//CasePacker.Status.Rate.Target := LREAL_TO_INT(csp_main_motorization_manager.motm.actual_velocity_setpoint);
//CasePacker.Status.Rate.Actual := LREAL_TO_INT(csp_main_motorization_manager.motm.actual_velocity);

//CasePacker.Status.Stop.AutoReason := csp_main_interface.alarm_id; 
//CasePacker.Status.Stop.Estop := machine_is_stop_emergency_active(csp.mch);
//CasePacker.Status.Stop.Guard := NOT safety_integrated_series_is_safely_closed(csp_case_main_safety_guards.sis) OR NOT safety_integrated_series_is_safely_closed(csp_transfer_main_safety_guards.sis);
//CasePacker.Status.Stop.Operator := message_is_on(csp_case_main_services_pushbuttons.stop_dchk.alarm_asm.message);

//CasePacker.Status.Starved.CaseBlanks := message_is_on(csp_case_feed_magazine_level_zonemin.magazine_level_zone_min_wem);
//CasePacker.Status.Starved.Glue := NOT digital_input_is_active(csp_case_glue_hotmelt.level_ok_di);
//CasePacker.Status.Starved.Labels :=
//CasePacker.Status.Starved.Units := csp_transfer_infeed_clamp.min_prime;

//CasePacker.Status.Blocked.Downstream := message_is_on(csp_case_discharge_reject_sensors.downstream_backup_hold_aem);
//CasePacker.Status.Blocked.Reject := message_is_on(csp_case_discharge_reject_sensors.consecutive_blocked_reject_aem);
//CasePacker.Status.Blocked.Waste := message_is_on(csp_transfer_crosspusher_reject.backup_di_dchk.alarm_asm.message);

//CasePacker.Labels.Consumed:=


(************************************************************************)

_handle_messages();

_write_output();

ACTION _handle_messages:
;
END_ACTION

ACTION _handle_process_test:
;
END_ACTION

ACTION _mode_manager:
IF process_mode_req_is_pending(prc)
THEN
    process_apply_mode_req_first_step(prc);
    CASE process_get_mode(prc) OF
        MODE_TO_ABSENT:
			;
        MODE_TO_INACTIVE:
			;
        MODE_TO_TEST:
			;
        MODE_TO_OPERATIONAL:
			;
    END_CASE
    process_apply_mode_req_second_step(prc);
END_IF
END_ACTION

ACTION _objects_manager:
IF objects_initialization()
THEN
	process_init(
		object_name					:= 'csp_customerInterfaces.prc', 
		machine						:= csp.mch, 
		CONVERSION_this				:= prc);
		
	prc_path 						:= process_get_path(prc);
END_IF

IF objects_running()
THEN
	process_cycle(prc);
END_IF
END_ACTION

ACTION _read_process_image:
;
END_ACTION

ACTION _read_var_input:
;
END_ACTION

ACTION _set_runtime_properties:
;
END_ACTION

ACTION _write_output:
;
END_ACTION

ACTION Dock:
//Flexlink to AMR Dock 1
CasePacker.Dock[1].DropAvailable:= csp_case_feed_magazine.Flexlink_to_AMR_DropAvailable_1;
CasePacker.Dock[1].PickAvailable:= csp_case_feed_magazine.Flexlink_to_AMR_PickAvailable_1; 
CasePacker.Dock[1].Active:= csp_case_feed_magazine.Flexlink_to_AMR_Active_1;
CasePacker.Dock[1].EntryAck:= csp_case_feed_magazine.Flexlink_to_AMR_EntryAck_1;
CasePacker.Dock[1].EntryOK:= csp_case_feed_magazine.Flexlink_to_AMR_EntryOK_1;

RAJ_to_Flexlink[3].0:= CasePacker.Dock[1].EntryReq;
RAJ_to_Flexlink[3].1:= CasePacker.Dock[1].AmrExited;

//Flexlink to AMR Dock 2
CasePacker.Dock[2].DropAvailable:= csp_case_feed_magazine.Flexlink_to_AMR_DropAvailable_2;
CasePacker.Dock[2].PickAvailable:= csp_case_feed_magazine.Flexlink_to_AMR_PickAvailable_2; 
CasePacker.Dock[2].Active:= csp_case_feed_magazine.Flexlink_to_AMR_Active_2;
CasePacker.Dock[2].EntryAck:= csp_case_feed_magazine.Flexlink_to_AMR_EntryAck_2;
CasePacker.Dock[2].EntryOK:= csp_case_feed_magazine.Flexlink_to_AMR_EntryOK_2;

RAJ_to_Flexlink[3].2:= CasePacker.Dock[2].EntryReq;
RAJ_to_Flexlink[3].3:= CasePacker.Dock[2].AmrExited;

//Flexlink to AMR Dock 3
CasePacker.Dock[3].DropAvailable:= csp_case_feed_magazine.Flexlink_to_AMR_DropAvailable_3;
CasePacker.Dock[3].PickAvailable:= csp_case_feed_magazine.Flexlink_to_AMR_PickAvailable_3; 
CasePacker.Dock[3].Active:= csp_case_feed_magazine.Flexlink_to_AMR_Active_3;
CasePacker.Dock[3].EntryAck:= csp_case_feed_magazine.Flexlink_to_AMR_EntryAck_3;
CasePacker.Dock[3].EntryOK:= csp_case_feed_magazine.Flexlink_to_AMR_EntryOK_3;

RAJ_to_Flexlink[3].4:= CasePacker.Dock[3].EntryReq;
RAJ_to_Flexlink[3].5:= CasePacker.Dock[3].AmrExited;
END_ACTION

END_PROGRAM

// ---- Application/CSP/Case/Feed/Magazine/csp_case_feed_magazine.TcPOU
(*********************************** G.D S.p.A. - Technical Department ***********************************
============= PROGRAM INFO ============
FOLDER:             TBD
MACHINES INVOLVED:  TBD 

============= DESCRIPTION =============
csp machine declaration

============= REVISIONS ===============
Date		Version	 	Author      	Description             
----------	-------		------------  	--------------------------------------------
2019/04/05 	0000.00	 	M.Grasso		Creation of the PRG

**********************************************************************************************************)
(*$R process_ref := prc; $*)
PROGRAM csp_case_feed_magazine
VAR
		
	prc:											process;
	prc_path:										STRING;
	
	
	
	
	AML_on_machine:									BOOL := true;
	Product_SKU:									DINT;
	Magazine_level_1:								DINT;
	AML_Load_Request:								BOOL;
	AML_loaded_holding_position:					BOOL;
	pusher_time_to_retract_timeout:					UDINT:= 20000; (* 20 seconds for rectract*)
	
	(* Signals From FLEXLINK *)
	AML_request_to_engage_pusher: 					BOOL := FALSE; //update _read_var_input
	AML_request_to_release_pusher:					BOOL := FALSE; ///update _read_var_input
	AML_Robot_Placing_Active:						BOOL := FALSE; //update _read_var_input with signal
	AML_Robot_Waiting_To_Place:						BOOL := FALSE; //update _read_var_input with signal
	AML_Robot_Out_Of_Cases:							BOOL := FALSE;//update _read_var_input with signal
	AML_Stop_Magazine_Conveyor:						BOOL := FALSE;//update _read_var_input with signal
	AML_Running:									BOOL := FALSE;//update _read_var_input with signal
	AML_Faulted:									BOOL := FALSE;//update _read_var_input with signal
	//Dock 1
	Flexlink_to_AMR_DropAvailable_1:				BOOL := FALSE;
	Flexlink_to_AMR_PickAvailable_1:				BOOL := FALSE;
	Flexlink_to_AMR_Active_1:						BOOL := FALSE;
	Flexlink_to_AMR_EntryAck_1:						BOOL := FALSE;
	Flexlink_to_AMR_EntryOK_1:						BOOL := FALSE;
	
	AMR_to_Flexlink_EntryReq_1:						BOOL := FALSE;
	AMR_to_Flexlink_AmrExited_1:					BOOL := FALSE;
	
	//Dock 2
	Flexlink_to_AMR_DropAvailable_2:				BOOL := FALSE;
	Flexlink_to_AMR_PickAvailable_2:				BOOL := FALSE;
	Flexlink_to_AMR_Active_2:						BOOL := FALSE;
	Flexlink_to_AMR_EntryAck_2:						BOOL := FALSE;
	Flexlink_to_AMR_EntryOK_2:						BOOL := FALSE;
	
	AMR_to_Flexlink_EntryReq_2:						BOOL := FALSE;
	AMR_to_Flexlink_AmrExited_2:					BOOL := FALSE;
	
	
	//Dock 3
	Flexlink_to_AMR_DropAvailable_3:				BOOL := FALSE;
	Flexlink_to_AMR_PickAvailable_3:				BOOL := FALSE;
	Flexlink_to_AMR_Active_3:						BOOL := FALSE;
	Flexlink_to_AMR_EntryAck_3:						BOOL := FALSE;
	Flexlink_to_AMR_EntryOK_3:						BOOL := FALSE;
	
	AMR_to_Flexlink_EntryReq_3:						BOOL := FALSE;
	AMR_to_Flexlink_AmrExited_3:					BOOL := FALSE;
	
	(* AML Messages For HMI *)
	AML_Robot_Faulted: 								message; 
	AML_Robot_Cases_Empty: 							message;
	AML_Robot_Loading_Cases_Active: 				message;
	AML_Request_To_Stop_Magazine_Conveyor: 			message;
	
	(* Signals TO FLEXLINK *)
	Pusher_Released: 								BOOL := FALSE;
	Ready_For_AML_Placement: 						BOOL := TRUE;
	Pusher_Engaged: 								BOOL := FALSE;
	Magazine_Level: 								BYTE;	(* Passed in from csp_case_feed_magazine_level, _read_var_input *)
	AML_Robot_Stop_Request:							BOOL := FALSE; //add logic to pass on stop request from CSP
	Case_Packer_Running:							BOOL := FALSE; //add logic to pass on running signal
	Case_Packer_Faulted:							BOOL := FALSE; //add logic to pass on faulted signal
	E_Stop_Channel_1_Open: 							BOOL := FALSE;
	E_Stop_Channel_2_Open: 							BOOL := FALSE;
	Guard_Zone_Channel_1_Open: 						BOOL := FALSE;
	Guard_Zone_Channel_2_Open: 						BOOL := FALSE;
	
	magazine_not_primed_motcond:					motorization_conditioner;
	
	
	toggle_button_input_di:							digital_input;
	toggle_button_led_do:							digital_output; (* 0 = OFF, 1 = ON *)
	toggle_button_color_do:							digital_output; (* 0 = GREEN, 1 = RED *)
	
	toggle_button_f_trig:							F_TRIG;
	toggle_button_input:							BOOL;
	
	toggle_button_ON:								BOOL;
	
	heart_beat: 									BOOL;
	test_pusher: 									BOOL;
	engage_delay: 									TON;
	Pusher_Engaged_Delayed: 						BOOL;
	
	magazine_disengage_enable:						BOOL:=FALSE;(*$P $*)
	AML_bypass_enable:								BOOL:=FALSE;(*$P $*)

	OS_mag_belt_ton: 								TON;
	OS_mag_belt_run_limit: 							BOOL;
	lS_mag_belt_ton: 								TON;
	lS_mag_belt_run_limit: 							BOOL;
	os_magazine_run_limit_aem: 						message;
	ls_magazine_run_limit_aem:						message;
	
	hold_request_aml_zone:							BOOL := FALSE;
	aml_zone_hold_motcond:							motorization_conditioner;
	aml_hold_bypass:								BOOL := FALSE;	
END_VAR

_read_var_input();

_object_manager();

IF NOT objects_running()
THEN
	RETURN;	
END_IF

_read_process_image();

_mode_manager();

_set_runtime_properties();

(********************************* BODY *********************************)

(* DETERMINES CONTROL OF MACHINE BASED ON AML PRESENCE OR MANUAL 8 BALL CONTROL *)
RAJ_to_Flexlink[0]:= Product_SKU;
RAJ_to_Flexlink[1] := Magazine_level;
RAJ_to_Flexlink[2].0:= Case_Packer_Running;
RAJ_to_Flexlink[2].1:= Case_Packer_Faulted;

RAJ_to_Flexlink[2].3:= Pusher_Released; 
RAJ_to_Flexlink[2].4:= Pusher_Engaged_Delayed;                                
RAJ_to_Flexlink[2].5:= Ready_For_AML_Placement;                         
RAJ_to_Flexlink[2].6:= csp_main_interface.Cartoner_RunOutRequest;                                  

RAJ_to_Flexlink[2].10 := heart_beat;
heart_beat := Flexlink_to_RAJ[2].10;
 
AML_request_to_engage_pusher:=Flexlink_to_RAJ[2].6;
AML_request_to_release_pusher:=Flexlink_to_RAJ[2].5;
AML_Robot_Placing_Active:=Flexlink_to_RAJ[2].7;
AML_Robot_Waiting_To_Place:=Flexlink_to_RAJ[2].2;
AML_Robot_Out_Of_Cases:=Flexlink_to_RAJ[2].3;
AML_Stop_Magazine_Conveyor:=Flexlink_to_RAJ[2].4;
AML_Running:=Flexlink_to_RAJ[2].0;
AML_Faulted:=Flexlink_to_RAJ[2].1;

//Flexlink to AMR bits dock 1
Flexlink_to_AMR_DropAvailable_1 := Flexlink_to_RAJ[3].0;
Flexlink_to_AMR_PickAvailable_1 := Flexlink_to_RAJ[3].1;					
Flexlink_to_AMR_Active_1 := Flexlink_to_RAJ[3].2;			
Flexlink_to_AMR_EntryAck_1 := Flexlink_to_RAJ[3].3;						
Flexlink_to_AMR_EntryOK_1 := Flexlink_to_RAJ[3].4;						

//RAJ_to_Flexlink[3].0 := AMR_to_Flexlink_EntryReq_1 ;	
//RAJ_to_Flexlink[3].1 := AMR_to_Flexlink_AmrExited_1;	

//Flexlink to AMR bits dock 2
Flexlink_to_AMR_DropAvailable_2 := Flexlink_to_RAJ[3].5;
Flexlink_to_AMR_PickAvailable_2 := Flexlink_to_RAJ[3].6;					
Flexlink_to_AMR_Active_2 := Flexlink_to_RAJ[3].7;			
Flexlink_to_AMR_EntryAck_2 := Flexlink_to_RAJ[3].8;						
Flexlink_to_AMR_EntryOK_2 := Flexlink_to_RAJ[3].9;						

//RAJ_to_Flexlink[3].2 := AMR_to_Flexlink_EntryReq_2 ;	
//RAJ_to_Flexlink[3].3 := AMR_to_Flexlink_AmrExited_2;

//Flexlink to AMR bits dock 3
Flexlink_to_AMR_DropAvailable_3 := Flexlink_to_RAJ[3].10;
Flexlink_to_AMR_PickAvailable_3 := Flexlink_to_RAJ[3].11;					
Flexlink_to_AMR_Active_3 := Flexlink_to_RAJ[3].12;			
Flexlink_to_AMR_EntryAck_3 := Flexlink_to_RAJ[3].13;						
Flexlink_to_AMR_EntryOK_3 := Flexlink_to_RAJ[3].14;						

//RAJ_to_Flexlink[3].4 := AMR_to_Flexlink_EntryReq_3 ;	
//RAJ_to_Flexlink[3].5 := AMR_to_Flexlink_AmrExited_3;

	
(*RAJ_to_Flexlink[0]:= Product_SKU;
		
RAJ_to_Flexlink[1] := Magazine_level_1;

Case_Packer_Running :=RAJ_to_Flexlink[2].1;*)


(* AML ACTIVE *)
IF AML_on_machine
THEN

	IF (
			csp_case_feed_magazine_level.level_status > CSP_CASE_FEED_MAGAZINE_LEVEL_STATUS_ZONE4 //Once we lose ZONE 4 PE, AML can request to load
			AND csp_main_services.pressure_switch_value > csp_main_services.pressure_value_limit //check pressure
			AND AML_request_to_release_pusher //input signal from FLEXLINK requesting to load
			AND NOT AML_request_to_engage_pusher
			AND NOT AML_bypass_enable //Links to button on main page that allows the the AML to be bypassed
		)	//input signal from Flexlink requesting to re-engage pushers
		OR csp_main_accuchange.Brand_Change_Occurred
	THEN
		AML_Load_Request := TRUE;
	ELSE
		AML_Load_Request := FALSE;
	END_IF
	
	hold_request_aml_zone := (AML_Stop_Magazine_Conveyor 
		OR digital_actuator_is_faulted(csp_case_feed_magazine_os_pusherTilt.sact)
		OR digital_actuator_is_faulted(csp_case_feed_magazine_ls_pusherTilt.sact))
		AND NOT aml_hold_bypass;
		
		
(* USING 8 BALL FOR CONTROL - AML NOT ACTIVE *)
ELSE
		
	toggle_button_f_trig(CLK := digital_input_is_active(toggle_button_input_di));
	toggle_button_input := toggle_button_f_trig.Q;

	IF csp_main_services.pressure_switch_value > csp_main_services.pressure_value_limit
	THEN
		digital_output_set(toggle_button_led_do);
		
		(* IF THE BUTTON IS PRESSED *)
		IF toggle_button_input
		THEN
			IF NOT toggle_button_ON
			THEN
				toggle_button_ON := TRUE;
			ELSE
				toggle_button_ON := FALSE;	
			END_IF
		END_IF		
	(* TURNS ON LED TEMPORARILY IF ACCU MAGAZINE AXIS IS MOVING *)
	ELSIF (axis_is_moving(csp_case_feed_magazine_accu_lsdepth.axis) OR axis_is_moving(csp_case_feed_magazine_accu_osdepth.axis))
	THEN
		digital_output_set(toggle_button_led_do);
 	ELSE
		digital_output_reset(toggle_button_led_do);
	END_IF
	
	
	(* CONTROLS LOAD REQUEST AND LED - INCLUDES ACCU AXIS MOVING *)
	IF toggle_button_ON
		OR (axis_is_moving(csp_case_feed_magazine_accu_lsdepth.axis) OR axis_is_moving(csp_case_feed_magazine_accu_osdepth.axis))
	THEN
		digital_output_set(toggle_button_color_do);
	ELSE
		digital_output_reset(toggle_button_color_do);
	END_IF
	
	IF toggle_button_ON
	THEN
		AML_Load_Request := TRUE;
	ELSE
		AML_Load_Request := FALSE;
	END_IF
END_IF

IF csp_main_services.pressure_switch_value > csp_main_services.pressure_value_limit //check pressure
	AND (digital_actuator_is_active(csp_case_feed_magazine_ls_pusher.sact)
	AND digital_actuator_is_active(csp_case_feed_magazine_os_pusher.sact)
	AND digital_actuator_is_active(csp_case_feed_magazine_ls_pusherTilt.sact)
	AND digital_actuator_is_active(csp_case_feed_magazine_os_pusherTilt.sact)
	AND csp_case_feed_magazine_ls_sensors.pusher_clear
	AND csp_case_feed_magazine_Os_sensors.pusher_clear)
	OR test_pusher
THEN
	Pusher_Released := TRUE; //AML in fully retracted position for LOAD
	Ready_For_AML_Placement := TRUE;
	Pusher_Engaged := FALSE;
ELSE
	Pusher_Engaged := TRUE;
	Ready_For_AML_Placement := TRUE;
	Pusher_Released := FALSE;
END_IF
	
engage_delay(IN:= Pusher_Engaged , PT:=T#5S , Q=> Pusher_Engaged_Delayed , ET=> );	

(* MAKES SURE THAT THE MAGAZINE THROAT PROXES ARE MET MEANING OK BACK PRESSURE FOR CASES *)
IF motorization_manager_is_starting(csp_main_motorization_manager.motm)
	AND filter_is_on(csp_case_feed_magazine_ls_sensors.feed_di_flt)
	AND filter_is_on(csp_case_feed_magazine_os_sensors.feed_di_flt)
	OR csp_case_main_services.dry_cycle_mode
THEN
	motorization_conditioner_start_done(magazine_not_primed_motcond);
END_IF

IF csp_main_services.pressure_switch_value > csp_main_services.pressure_value_limit //check pressure
THEN
	digital_actuator_message_enable(csp_case_feed_magazine_ls_pusher.sact);
	digital_actuator_message_enable(csp_case_feed_magazine_os_pusher.sact);
	digital_actuator_message_enable(csp_case_feed_magazine_ls_pushertilt.sact);
	digital_actuator_message_enable(csp_case_feed_magazine_os_pusherTilt.sact);
ELSE
	digital_actuator_message_disable(csp_case_feed_magazine_ls_pusher.sact);
	digital_actuator_message_disable(csp_case_feed_magazine_os_pusher.sact);
	digital_actuator_message_disable(csp_case_feed_magazine_ls_pushertilt.sact);
	digital_actuator_message_disable(csp_case_feed_magazine_os_pusherTilt.sact);
END_IF

OS_mag_belt_ton(IN:= axis_is_moving(csp_case_feed_magazine_os_belt.axis) , PT:=T#5S , Q=> OS_mag_belt_run_limit , ET=> );		
lS_mag_belt_ton(IN:= axis_is_moving(csp_case_feed_magazine_ls_belt.axis) , PT:=T#5S , Q=> lS_mag_belt_run_limit , ET=> );

IF	OS_mag_belt_run_limit
THEN
	process_message_set(0, 0, 0, os_magazine_run_limit_aem);
ELSE
	process_message_reset(os_magazine_run_limit_aem);	
END_IF

IF	LS_mag_belt_run_limit
THEN
	process_message_set(0, 0, 0, ls_magazine_run_limit_aem);
ELSE
		process_message_reset(ls_magazine_run_limit_aem);	
END_IF

IF	hold_request_aml_zone
	AND NOT aml_hold_bypass
	AND csp_main_motorization_manager.debug_Enable_new_conditioners (* Selector on HMI while still being tested *)
THEN
	motorization_conditioner_hold(aml_zone_hold_motcond);
	motorization_conditioner_velocity_limit_activate(aml_zone_hold_motcond);
ELSE
	motorization_conditioner_unhold(aml_zone_hold_motcond);
	motorization_conditioner_velocity_limit_deactivate(aml_zone_hold_motcond);
END_IF

(************************************************************************)

_handle_messages();

_write_output();

ACTION _handle_messages:
IF AML_Faulted 
THEN
	process_message_set(0,0,0,AML_Robot_Faulted);
ELSE
	Process_message_reset(AML_Robot_Faulted);
END_IF


IF AML_Robot_Out_Of_Cases
THEN
	process_message_set(0,0,0,AML_Robot_Cases_Empty);
ELSE
	process_message_reset(AML_Robot_Cases_Empty);
END_IF

IF AML_Robot_Placing_Active
THEN
	process_message_set(0,0,0, AML_Robot_Loading_Cases_Active);
ELSE
	process_message_reset(AML_Robot_Loading_Cases_Active);
END_IF

IF AML_Stop_Magazine_Conveyor
THEN
	process_message_set(0,0,0, AML_Request_To_Stop_Magazine_Conveyor);
ELSE
	process_message_reset(AML_Request_To_Stop_Magazine_Conveyor);
END_IF



;
END_ACTION

ACTION _handle_process_test:
;
END_ACTION

ACTION _mode_manager:
IF process_mode_req_is_pending(prc)
THEN
    process_apply_mode_req_first_step(prc);
    CASE process_get_mode(prc) OF
        MODE_TO_ABSENT:
			;
        MODE_TO_INACTIVE:
			;
        MODE_TO_TEST:
			;
        MODE_TO_OPERATIONAL:
			;
    END_CASE
    process_apply_mode_req_second_step(prc);
END_IF
END_ACTION

ACTION _object_manager:
IF objects_initialization()
THEN
	sub_process_init(
		object_name					:= 'csp_case_feed_magazine.prc', 
		process						:= csp_case_feed.prc, 
		CONVERSION_this				:= prc);
		
	prc_path 						:= process_get_path(prc);
	
	process_message_init(
        object_name:= CONCAT(prc_path, 'AML_Robot_Faulted'),
        behaviour:= MESSAGE_BEHAVIOUR_STATE,
        reset_timeout:= 0,
        disableable:= TRUE,
        individual_reset:= FALSE,
        machine_reaction:= MACHINE_REACTION_NO_STOP, 
        typology:=  MESSAGE_TYPOLOGY_OBLIGATION,
        process:= prc,
        CONVERSION_this:= AML_Robot_Faulted);
		
	process_message_init(
        object_name:= CONCAT(prc_path, 'AML_Robot_Cases_Empty'),
        behaviour:= MESSAGE_BEHAVIOUR_STATE,
        reset_timeout:= 0,
        disableable:= TRUE,
        individual_reset:= FALSE,
        machine_reaction:= MACHINE_REACTION_NO_STOP, 
        typology:=  MESSAGE_TYPOLOGY_OBLIGATION,
        process:= prc,
        CONVERSION_this:= AML_Robot_Cases_Empty);

	process_message_init(
        object_name:= CONCAT(prc_path, 'AML_Robot_Loading_Cases_Active'),
        behaviour:= MESSAGE_BEHAVIOUR_STATE,
        reset_timeout:= 0,
        disableable:= TRUE,
        individual_reset:= FALSE,
        machine_reaction:= MACHINE_REACTION_NO_STOP,
        typology:=  MESSAGE_TYPOLOGY_NORMAL,
        process:= prc,
        CONVERSION_this:= AML_Robot_Loading_Cases_Active);
		
	process_message_init(
        object_name:= CONCAT(prc_path, 'AML_Request_To_Stop_Magazine_Conveyor'),
        behaviour:= MESSAGE_BEHAVIOUR_STATE,
        reset_timeout:= 0,
        disableable:= TRUE,
        individual_reset:= FALSE,
        machine_reaction:= MACHINE_REACTION_NO_STOP,
        typology:=  MESSAGE_TYPOLOGY_OBLIGATION, 
        process:= prc,
        CONVERSION_this:= AML_Request_To_Stop_Magazine_Conveyor);
	
	motorization_conditioner_init(
		object_name					:=	CONCAT(prc_path, '_magazine_not_primed_motcond'),
		velocity_limit				:=	0.0,
		velocity_limit_active		:=	FALSE,
		idle_handshake_active		:=	FALSE,
		execute_handshake_active	:=	TRUE,
		hold_handshake_active		:=	FALSE,
		suspend_handshake_active	:=	FALSE,
		complete_handshake_active	:=	FALSE,
		abort_handshake_active		:=	FALSE,
		stop_handshake_active		:=	FALSE,
		origin						:=	MOTORIZATION_CONDITIONER_ORIGIN_INTERNAL,
		manager						:=	csp_main_motorization_manager.motm,
		process						:=	prc,
		CONVERSION_this				:=	magazine_not_primed_motcond);
	
	
	(* OUTPUTS *)
	digital_output_init(
		object_name 			:= CONCAT(prc_path, '_toggle_button_led_do'),
		polarity_direct 		:= TRUE,
		process 				:= prc,
		CONVERSION_this 		:= toggle_button_led_do);
		
	digital_output_init(
		object_name 			:= CONCAT(prc_path, '_toggle_button_color_do'),
		polarity_direct 		:= TRUE,
		process 				:= prc,
		CONVERSION_this 		:= toggle_button_color_do);
		
	(* INPUTS *) 
	digital_input_init(
		object_name					:= CONCAT(prc_path, '_toggle_button_input_di'), 
		polarity_direct				:= TRUE, 
		process						:= prc, 
		CONVERSION_this				:= toggle_button_input_di);
		
	process_message_init(
		object_name:= CONCAT(prc_path, '_os_magazine_run_limit_aem'), 
		behaviour:= MESSAGE_BEHAVIOUR_EVENT, 
		reset_timeout:= 0, 
		disableable:= FALSE, 
		individual_reset:= FALSE, 
		machine_reaction:= MACHINE_REACTION_STOP_IN_PHASE_ONE, 
		typology:= MESSAGE_TYPOLOGY_ABNORMAL, 
		process:= prc, 
		CONVERSION_this:= os_magazine_run_limit_aem);	
		
	process_message_init(
		object_name:= CONCAT(prc_path, '_ls_magazine_run_limit_aem'), 
		behaviour:= MESSAGE_BEHAVIOUR_EVENT, 
		reset_timeout:= 0, 
		disableable:= FALSE, 
		individual_reset:= FALSE, 
		machine_reaction:= MACHINE_REACTION_STOP_IN_PHASE_ONE, 
		typology:= MESSAGE_TYPOLOGY_ABNORMAL, 
		process:= prc, 
		CONVERSION_this:= ls_magazine_run_limit_aem);	
	
	motorization_conditioner_init(
		object_name := CONCAT(prc_path, '_aml_zone_hold_motcond'),
		velocity_limit := 0,
		velocity_limit_active := FALSE,
		idle_handshake_active := FALSE,
		execute_handshake_active := FALSE,
		hold_handshake_active := FALSE,
		suspend_handshake_active := FALSE,
		complete_handshake_active := FALSE,
		abort_handshake_active := FALSE,
		stop_handshake_active := FALSE,
		origin := MOTORIZATION_CONDITIONER_ORIGIN_EXTERNAL_UP,
		manager := csp_main_motorization_manager.motm,
		process := prc,
		CONVERSION_this := aml_zone_hold_motcond);
	
END_IF

IF objects_running()
THEN
	process_cycle(prc);
	motorization_conditioner_cycle(magazine_not_primed_motcond);
	motorization_conditioner_cycle(aml_zone_hold_motcond);

END_IF
END_ACTION

ACTION _read_process_image:
;
END_ACTION

ACTION _read_var_input:
//AML_request_to_engage_pusher 		:= input FROM flexlink;
//AML_request_to_release_pusher 	:= input FROM flexlink;
//AML_Robot_Placing_Active 			:= input from Flexlink;
//AML_Robot_Waiting_To_Place 		:= input from flexlink;
//AML_Robot_Out_Of_Cases 			:= input from flexlink;				
//AML_Stop_Magazine_Conveyor 		:= input from flexlink;					
//AML_Running 						:= input from flexlink;					
//AML_Faulted 						:= input from flexlink;
//AML_E_Stop_Channel_1_Open			:= input FROM flexlink;
//AML_E_Stop_Channel_2_Open			:= input FROM flexlink;
//AML_Guard_Zone_Channel_1_Open		:= input from flexlink;
//AML_Guard_Zone_Channel_2_Open		:= input from flexlink;

Magazine_Level := csp_case_feed_magazine_level.level;


(* Add Logic to get this information AMR *)

//AML_Robot_Stop_Request := //add logic to pass on stop request from CSP
Case_Packer_Running := machine_is_execute(csp.mch);	//add logic to pass on running signal
Case_Packer_Faulted := machine_is_stopped(csp.mch); //add logic to pass on faulted signal	
E_Stop_Channel_1_Open := safety_integrated_object_protection_is_open(csp_case_main_safety_emergency.HMI_button_sio);
E_Stop_Channel_2_Open := safety_integrated_object_protection_is_open(csp_transfer_main_safety_emergency.HMI_button_sio);
Guard_Zone_Channel_1_Open := NOT safety_integrated_series_is_safely_closed(csp_case_main_safety_guards.sis);		
Guard_Zone_Channel_2_Open := NOT safety_integrated_series_is_safely_closed(csp_transfer_main_safety_guards.sis);	

						
;
END_ACTION

ACTION _set_runtime_properties:
;
END_ACTION

ACTION _write_output:
;
END_ACTION

END_PROGRAM

// ---- Application/CSP/Main/Phase Manager/csp_main_phaseManager_startJob.TcPOU
(*********************************** G.D S.p.A. - Technical Department ***********************************
============= PROGRAM INFO ============
FOLDER:             TBD
MACHINES INVOLVED:  TBD 

============= DESCRIPTION =============
WU phase manager program

============= REVISIONS ===============
Date		Version	 	Author      	Description             
----------	-------		------------  	--------------------------------------------
2020/06/16 	0000.00	 	G.Cera 			Creation of the PRG
2021/01/08 	0000.01	 	S.Uccellari 	Filler version
**********************************************************************************************************)
(*$R
	process_ref := prc;
$*)
PROGRAM csp_main_phaseManager_startJob
VAR
	prc:												process;
	prc_path:											STRING;
	
	fsm_enable_conditions:								BOOL;
	fsm_status:											INT;
	
	index:												INT;
	
	start_job_running:									BOOL;
	start_job_done:										BOOL;
	start_job_in_progress_wsm:							message;
	start_job_in_progress_asm:							message;
	machine_setup_in_progress_wsm:						message;
	
	execute_machine_setup:								BOOL := TRUE; (*MARCO - temporary*)
	machine_setup_completed_bor:						boolean_or;

	check_MES_variables:								BOOL;
	MES_variables_valid:								BOOL;
	
	check_order_information:							BOOL;
	order_valid:										BOOL;

	check_product_information:							BOOL;
	product_valid:										BOOL;
	cups_number_valid:									BOOL;

	check_recipe_information:							BOOL;
	recipe_valid:										BOOL;
	
	check_curr_material_information:					BOOL;
	curr_material_valid:								BOOL;
		
	check_next_material_information:					BOOL;
	next_material_valid:								BOOL;
			
	check_mark_bubd_information:						BOOL;
	mark_bubd_valid:									BOOL;

	order_valid_led:									led;	
	product_valid_led:									led;	
	recipe_valid_led:									led;	
	materials_valid_led:								led;	
	mark_valid_led:										led;	
	
	order_ID:											STRING;												(*$M $*)
	order_SAP_batch_ID:									STRING;												(*$M $*)

	product_ID:											STRING;												(*$M $*)
	product_UPC:										STRING;												(*$M $*)
	product_pods_per_carton:							INT;												(*$M $*)
	product_pods_per_case:								INT;												(*$M $*)
	product_cartons_per_case:							INT;												(*$M $*)
	product_target_weight:								REAL;												(*$M $*)
	product_min_weight:									REAL;												(*$M $*)
	product_max_weight:									REAL;												(*$M $*)
	product_filter_type:								STRING;												(*$M $*)
	caffeinated_flag_led:								led;
	kosher_flag_led:									led;
	organic_flag_led:									led;
	flavor_flag_led:									led;
	product_flavor_dose:								REAL;												(*$M $*)
	product_shelf_life:									INT;												(*$M $*)
	
	recipe_filler:										STRING;												(*$M $*)
	recipe_cartoner:									STRING;												(*$M $*)
	recipe_case_packer:									STRING;												(*$M $*)
	
	current_material_1_ID:								STRING;												(*$M $*)
	current_material_1_QTY:								REAL;												(*$M $*)
	current_material_2_ID:								STRING;												(*$M $*)
	current_material_2_QTY:								REAL;												(*$M $*)
	current_material_3_ID:								STRING;												(*$M $*)
	current_material_3_QTY:								REAL;												(*$M $*)
	current_material_4_ID:								STRING;												(*$M $*)
	current_material_4_QTY:								REAL;												(*$M $*)
	current_material_5_ID:								STRING;												(*$M $*)
	current_material_5_QTY:								REAL;												(*$M $*)
	current_material_6_ID:								STRING;												(*$M $*)
	current_material_6_QTY:								REAL;												(*$M $*)
	current_material_7_ID:								STRING;												(*$M $*)
	current_material_7_QTY:								REAL;												(*$M $*)
	current_material_8_ID:								STRING;												(*$M $*)
	current_material_8_QTY:								REAL;												(*$M $*)
	current_material_9_ID:								STRING;												(*$M $*)
	current_material_9_QTY:								REAL;												(*$M $*)
	current_material_10_ID:								STRING;												(*$M $*)
	current_material_10_QTY:							REAL;												(*$M $*)
	current_material_11_ID:								STRING;												(*$M $*)
	current_material_11_QTY:							REAL;												(*$M $*)
	current_material_12_ID:								STRING;												(*$M $*)
	current_material_12_QTY:							REAL;												(*$M $*)
	current_material_13_ID:								STRING;												(*$M $*)
	current_material_13_QTY:							REAL;												(*$M $*)
	current_material_14_ID:								STRING;												(*$M $*)
	current_material_14_QTY:							REAL;												(*$M $*)
	current_material_15_ID:								STRING;												(*$M $*)
	current_material_15_QTY:							REAL;												(*$M $*)

	next_material_1_ID:									STRING;												(*$M $*)
	next_material_1_QTY:								REAL;												(*$M $*)
	next_material_2_ID:									STRING;												(*$M $*)
	next_material_2_QTY:								REAL;												(*$M $*)
	next_material_3_ID:									STRING;												(*$M $*)
	next_material_3_QTY:								REAL;												(*$M $*)
	next_material_4_ID:									STRING;												(*$M $*)
	next_material_4_QTY:								REAL;												(*$M $*)
	next_material_5_ID:									STRING;												(*$M $*)
	next_material_5_QTY:								REAL;												(*$M $*)
	next_material_6_ID:									STRING;												(*$M $*)
	next_material_6_QTY:								REAL;												(*$M $*)
	next_material_7_ID:									STRING;												(*$M $*)
	next_material_7_QTY:								REAL;												(*$M $*)
	next_material_8_ID:									STRING;												(*$M $*)
	next_material_8_QTY:								REAL;												(*$M $*)
	next_material_9_ID:									STRING;												(*$M $*)
	next_material_9_QTY:								REAL;												(*$M $*)
	next_material_10_ID:								STRING;												(*$M $*)
	next_material_10_QTY:								REAL;												(*$M $*)
	next_material_11_ID:								STRING;												(*$M $*)
	next_material_11_QTY:								REAL;												(*$M $*)
	next_material_12_ID:								STRING;												(*$M $*)
	next_material_12_QTY:								REAL;												(*$M $*)
	next_material_13_ID:								STRING;												(*$M $*)
	next_material_13_QTY:								REAL;												(*$M $*)
	next_material_14_ID:								STRING;												(*$M $*)
	next_material_14_QTY:								REAL;												(*$M $*)
	next_material_15_ID:								STRING;												(*$M $*)
	next_material_15_QTY:								REAL;												(*$M $*)
	
	mark_BUBD:											STRING;												(*$M $*)
	mark_prefix:										STRING;												(*$M $*)
	mark_format:										STRING;												(*$M $*)
	
	i_end_job_done:										POINTER TO BOOL;	
	
	debug_mes_startJobReq:								BOOL;
	debug_mes_cycleEnable:								BOOL;		
	
END_VAR

VAR PERSISTENT
	order_information:									csp_customerInterfaces_order;
	product_information:								csp_customerInterfaces_product;
	recipe_information:									csp_customerInterfaces_recipe;
	current_material_information:						ARRAY[0..14] OF csp_customerInterfaces_material;
	next_material_information:							ARRAY[0..14] OF csp_customerInterfaces_material;
	mark_bubd_information:								csp_customerInterfaces_markBUBD;
END_VAR

_read_var_input();

_object_manager();

IF NOT objects_running()
THEN
	RETURN;	
END_IF

_read_process_image();

_mode_manager();

CASE process_get_mode(prc) of
	MODE_ABSENT,
	MODE_INACTIVE:
		RETURN;
	MODE_TEST:
		_handle_process_test();
END_CASE

_set_runtime_properties();

(********************************* BODY *********************************)

(************************************************************************)

(**************************** PROGRAM HANDLER ***************************)
run_cycle();
check_parameters();
custom_page();
(************************************************************************)

_handle_messages();

_write_output();

ACTION _handle_messages:
IF	(
		csp_main_phaseManager.fsm_status
		=
		CSP_MAIN_PHASE_MANAGER_STATUS_START_JOB_10
	)
THEN
	IF 	execute_machine_setup
	THEN	
		process_message_set(
			errorID_1			:= 1, 
			errorID_2			:= 0, 
			errorID_3			:= 0, 
			CONVERSION_this		:= start_job_in_progress_wsm);

		//process_message_reset(start_job_in_progress_asm);
	ELSE
		(*process_message_set(
			errorID_1			:= 1, 
			errorID_2			:= 0, 
			errorID_3			:= 0, 
			CONVERSION_this		:= start_job_in_progress_asm);
		*)
		process_message_reset(start_job_in_progress_wsm);	
	END_IF	
ELSE
	process_message_reset(start_job_in_progress_wsm);	
	//process_message_reset(start_job_in_progress_asm);		
END_IF

(*
IF 	execute_machine_setup
THEN
	process_message_set(
		errorID_1			:= 1, 
		errorID_2			:= 0, 
		errorID_3			:= 0, 
		CONVERSION_this		:= machine_setup_in_progress_wsm);
ELSE
	process_message_reset(machine_setup_in_progress_wsm);
END_IF
*)
END_ACTION

ACTION _handle_process_test:
;
END_ACTION

ACTION _mode_manager:
IF process_mode_req_is_pending(prc)
THEN
    process_apply_mode_req_first_step(prc);
    CASE process_get_mode(prc) OF
        MODE_TO_ABSENT:
			;
        MODE_TO_INACTIVE:
			;
        MODE_TO_TEST:
			;
        MODE_TO_OPERATIONAL:
			;
    END_CASE
    process_apply_mode_req_second_step(prc);
END_IF
END_ACTION

ACTION _object_manager:
IF objects_initialization()
THEN
	sub_process_init(
		object_name					:= 'csp_main_phaseManager_startJob.prc', 
		process						:= csp_main_phaseManager.prc, 
		CONVERSION_this				:= prc);
		
	prc_path 						:= process_get_path(prc);
	
	boolean_or_init(
		object_name					:= CONCAT(prc_path, '_machine_setup_completed_bor'), 
		process						:= prc, 
		CONVERSION_this				:= machine_setup_completed_bor);

	led_init(
		object_name					:= CONCAT(prc_path, '_caffeinated_flag_led'), 
		process						:= prc, 
		CONVERSION_this				:= caffeinated_flag_led);		
		
	led_init(
		object_name					:= CONCAT(prc_path, '_kosher_flag_led'), 
		process						:= prc, 
		CONVERSION_this				:= kosher_flag_led);	

	led_init(
		object_name					:= CONCAT(prc_path, '_organic_flag_led'), 
		process						:= prc, 
		CONVERSION_this				:= organic_flag_led);	

	led_init(
		object_name					:= CONCAT(prc_path, '_flavor_flag_led'), 
		process						:= prc, 
		CONVERSION_this				:= flavor_flag_led);				
		
	led_init(
		object_name					:= CONCAT(prc_path, '_order_valid_led'), 
		process						:= prc, 
		CONVERSION_this				:= order_valid_led);
		
	led_init(
		object_name					:= CONCAT(prc_path, '_product_valid_led'), 
		process						:= prc, 
		CONVERSION_this				:= product_valid_led);

	led_init(
		object_name					:= CONCAT(prc_path, '_recipe_valid_led'), 
		process						:= prc, 
		CONVERSION_this				:= recipe_valid_led);	

	led_init(
		object_name					:= CONCAT(prc_path, '_materials_valid_led'), 
		process						:= prc, 
		CONVERSION_this				:= materials_valid_led);

	led_init(
		object_name					:= CONCAT(prc_path, '_mark_valid_led'), 
		process						:= prc, 
		CONVERSION_this				:= mark_valid_led);				
		
	process_message_init(
		object_name					:= CONCAT(prc_path, '_start_job_in_progress_asm'), 
		behaviour					:= MESSAGE_BEHAVIOUR_TRY_AND_CHECK, 
		reset_timeout				:= 5000, 
		disableable					:= FALSE, 
		individual_reset			:= FALSE, 
		machine_reaction			:= MACHINE_REACTION_NORMAL_STOP, 
		typology					:= MESSAGE_TYPOLOGY_ABNORMAL, 
		process						:= prc, 
		CONVERSION_this				:= start_job_in_progress_asm);	
		
	process_message_init(
		object_name					:= CONCAT(prc_path, '_start_job_in_progress_wsm'), 
		behaviour					:= MESSAGE_BEHAVIOUR_TRY_AND_CHECK, 
		reset_timeout				:= 5000, 
		disableable					:= FALSE, 
		individual_reset			:= FALSE, 
		machine_reaction			:= MACHINE_REACTION_NO_STOP, 
		typology					:= MESSAGE_TYPOLOGY_NORMAL, 
		process						:= prc, 
		CONVERSION_this				:= start_job_in_progress_wsm);			
		
	process_message_init(
		object_name					:= CONCAT(prc_path, '_machine_setup_in_progress_wsm'), 
		behaviour					:= MESSAGE_BEHAVIOUR_TRY_AND_CHECK, 
		reset_timeout				:= 5000, 
		disableable					:= FALSE, 
		individual_reset			:= FALSE, 
		machine_reaction			:= MACHINE_REACTION_NO_STOP, 
		typology					:= MESSAGE_TYPOLOGY_NORMAL, 
		process						:= prc, 
		CONVERSION_this				:= machine_setup_in_progress_wsm);		
		
	
		
END_IF

IF objects_running()
THEN
	process_cycle(prc);
END_IF
END_ACTION

ACTION _read_process_image:
;
END_ACTION

ACTION _read_var_input:
i_end_job_done := ADR(csp_main_phaseManager_end_job.end_job_done);
END_ACTION

ACTION _set_runtime_properties:
;
END_ACTION

ACTION _write_output:
;
END_ACTION

ACTION check_parameters:
IF NOT start_job_running
THEN
	order_valid := FALSE;
	product_valid := FALSE;
	recipe_valid := FALSE;
	curr_material_valid := FALSE;
	next_material_valid := FALSE;
	mark_bubd_valid := FALSE;
END_IF

IF	check_MES_variables
THEN
// Order variable check
	IF 	(
			order_information.ID
			<>
			''
		)
		AND
		(
			order_information.SapBatchID
			<>
			''
		)
	THEN
		order_valid := TRUE;
	ELSE
		
		order_valid := FALSE;
	END_IF	

// Product variable check	
	IF 	product_information.ID <> ''
		AND
			product_information.UPC <> ''
		AND
			product_information.PodsPerCarton > 0
		AND
			product_information.PodsPerCase > 0
		AND
			product_information.ShelfLife > 0
		AND		
		(	product_information.FillWeight.Maximum > product_information.FillWeight.Target
			AND
			product_information.FillWeight.Target > product_information.FillWeight.Minimum
			AND
			product_information.FillWeight.Minimum > 0	)
		AND
		(	product_information.FilterType = 'LFF'
			OR
			product_information.FilterType = 'FLUT'	)
	THEN
		product_valid := TRUE;
	ELSE		
		product_valid := FALSE;
	END_IF	

// Recipe variable check	
	IF	recipe_information.Filler
		<>
		''
	THEN
		recipe_valid := TRUE;
	ELSE
		recipe_valid := FALSE;
	END_IF	

// Current material variable check	
	curr_material_valid := TRUE;
	
	IF	current_material_information[csp_main_phaseManager.MASTER_CASE_BLANK_MATERIAL_ID].ID = ''
	THEN
		curr_material_valid := FALSE;
	END_IF
	IF	(	current_material_information[csp_main_phaseManager.MASTER_CASE_BLANK_MATERIAL_ID].ID <> 'None' 
			AND
			current_material_information[csp_main_phaseManager.MASTER_CASE_BLANK_MATERIAL_ID].QTY = 0	)
		OR
		(	current_material_information[csp_main_phaseManager.MASTER_CASE_BLANK_MATERIAL_ID].ID <> 'None' 
			AND
			current_material_information[csp_main_phaseManager.MASTER_CASE_BLANK_MATERIAL_ID].QTY <= 0	)
	THEN
		curr_material_valid := FALSE;
	END_IF

	(*
	IF	current_material_information[csp_main_phaseManager.CASE_LABEL_MATERIAL_ID].ID = ''
	THEN
		curr_material_valid := FALSE;
	END_IF
	IF	(	current_material_information[csp_main_phaseManager.CASE_LABEL_MATERIAL_ID].ID <> 'None' 
			AND
			current_material_information[csp_main_phaseManager.CASE_LABEL_MATERIAL_ID].QTY = 0	)
		OR
		(	current_material_information[csp_main_phaseManager.CASE_LABEL_MATERIAL_ID].ID <> 'None' 
			AND
			current_material_information[csp_main_phaseManager.CASE_LABEL_MATERIAL_ID].QTY <= 0	)
	THEN
		curr_material_valid := FALSE;
	END_IF
	*)
	
// Next material variable check	
	next_material_valid := TRUE;

	IF	next_material_information[csp_main_phaseManager.MASTER_CASE_BLANK_MATERIAL_ID].ID = ''
	THEN
		next_material_valid := FALSE;
	END_IF
	IF	(	next_material_information[csp_main_phaseManager.MASTER_CASE_BLANK_MATERIAL_ID].ID <> 'None' 
			AND
			next_material_information[csp_main_phaseManager.MASTER_CASE_BLANK_MATERIAL_ID].QTY = 0	)
		OR
		(	next_material_information[csp_main_phaseManager.MASTER_CASE_BLANK_MATERIAL_ID].ID <> 'None' 
			AND
			next_material_information[csp_main_phaseManager.MASTER_CASE_BLANK_MATERIAL_ID].QTY <= 0	)
	THEN
		next_material_valid := FALSE;
	END_IF

(*		
	IF	next_material_information[csp_main_phaseManager.CASE_LABEL_MATERIAL_ID].ID = ''
	THEN
		next_material_valid := FALSE;
	END_IF
	IF	(	next_material_information[csp_main_phaseManager.CASE_LABEL_MATERIAL_ID].ID <> 'None' 
			AND
			next_material_information[csp_main_phaseManager.CASE_LABEL_MATERIAL_ID].QTY = 0	)
		OR
		(	next_material_information[csp_main_phaseManager.CASE_LABEL_MATERIAL_ID].ID <> 'None' 
			AND
			next_material_information[csp_main_phaseManager.CASE_LABEL_MATERIAL_ID].QTY <= 0	)
	THEN
		next_material_valid := FALSE;
	END_IF
*)
	
// Mark BUBD variable check
	IF	(
			mark_bubd_information.BestUsedByDate
			<>
			''
		)
		AND
		(
			mark_bubd_information.Prefix
			<>
			''
		)
	THEN
		mark_bubd_valid := TRUE;
	ELSE
		mark_bubd_valid := FALSE;
	END_IF	
END_IF

MES_variables_valid :=
	order_valid
	AND
	product_valid
	AND
	recipe_valid
	AND
	curr_material_valid
	(*AND
	next_material_valid*)
	AND
	mark_bubd_valid;
END_ACTION

ACTION custom_page:
order_ID := order_information.ID;
order_SAP_batch_ID := order_information.SapBatchID;

product_ID := product_information.ID;
product_UPC := product_information.UPC;
product_pods_per_carton := product_information.PodsPerCarton;
product_pods_per_case := product_information.PodsPerCase;
product_cartons_per_case := product_information.CartonsPerCase;
product_target_weight := product_information.FillWeight.Target;
product_min_weight := product_information.FillWeight.Minimum;
product_max_weight := product_information.FillWeight.Maximum;
product_filter_type := product_information.FilterType;
product_flavor_dose := product_information.FlavorDose;
product_shelf_life := product_information.ShelfLife;

IF	product_information.CaffeinatedFlag
THEN
	led_set_color(
		color				:= HMI_LED_COLOR_GREEN, 
		CONVERSION_this		:= caffeinated_flag_led);	
ELSE
	led_set_color(
		color				:= HMI_LED_COLOR_RED, 
		CONVERSION_this		:= caffeinated_flag_led);	
END_IF

IF	product_information.KosherFlag
THEN
	led_set_color(
		color				:= HMI_LED_COLOR_GREEN, 
		CONVERSION_this		:= kosher_flag_led);	
ELSE
	led_set_color(
		color				:= HMI_LED_COLOR_RED, 
		CONVERSION_this		:= kosher_flag_led);	
END_IF

IF	product_information.OrganicFlag
THEN
	led_set_color(
		color				:= HMI_LED_COLOR_GREEN, 
		CONVERSION_this		:= organic_flag_led);	
ELSE
	led_set_color(
		color				:= HMI_LED_COLOR_RED, 
		CONVERSION_this		:= organic_flag_led);	
END_IF

IF	product_information.FlavorFlag
THEN
	led_set_color(
		color				:= HMI_LED_COLOR_GREEN, 
		CONVERSION_this		:= flavor_flag_led);	
ELSE
	led_set_color(
		color				:= HMI_LED_COLOR_RED, 
		CONVERSION_this		:= flavor_flag_led);	
END_IF

recipe_filler := recipe_information.Filler;
recipe_cartoner := recipe_information.Cartoner;
recipe_case_packer := recipe_information.CasePacker;

current_material_1_ID := current_material_information[0].ID;
current_material_1_QTY := current_material_information[0].QTY;
current_material_2_ID := current_material_information[1].ID;
current_material_2_QTY := current_material_information[1].QTY;
current_material_3_ID := current_material_information[2].ID;
current_material_3_QTY := current_material_information[2].QTY;
current_material_4_ID := current_material_information[3].ID;
current_material_4_QTY := current_material_information[3].QTY;
current_material_5_ID := current_material_information[4].ID;
current_material_5_QTY := current_material_information[4].QTY;
current_material_6_ID := current_material_information[5].ID;
current_material_6_QTY := current_material_information[5].QTY;
current_material_7_ID := current_material_information[6].ID;
current_material_7_QTY := current_material_information[6].QTY;
current_material_8_ID := current_material_information[7].ID;
current_material_8_QTY := current_material_information[7].QTY;
current_material_9_ID := current_material_information[8].ID;
current_material_9_QTY := current_material_information[8].QTY;
current_material_10_ID := current_material_information[9].ID;
current_material_10_QTY := current_material_information[9].QTY;
current_material_11_ID := current_material_information[10].ID;
current_material_11_QTY := current_material_information[10].QTY;
current_material_12_ID := current_material_information[11].ID;
current_material_12_QTY := current_material_information[11].QTY;
current_material_13_ID := current_material_information[12].ID;
current_material_13_QTY := current_material_information[12].QTY;
current_material_14_ID := current_material_information[13].ID;
current_material_14_QTY := current_material_information[13].QTY;
current_material_15_ID := current_material_information[14].ID;
current_material_15_QTY := current_material_information[14].QTY;

next_material_1_ID := next_material_information[0].ID;
next_material_1_QTY := next_material_information[0].QTY;
next_material_2_ID := next_material_information[1].ID;
next_material_2_QTY := next_material_information[1].QTY;
next_material_3_ID := next_material_information[2].ID;
next_material_3_QTY := next_material_information[2].QTY;
next_material_4_ID := next_material_information[3].ID;
next_material_4_QTY := next_material_information[3].QTY;
next_material_5_ID := next_material_information[4].ID;
next_material_5_QTY := next_material_information[4].QTY;
next_material_6_ID := next_material_information[5].ID;
next_material_6_QTY := next_material_information[5].QTY;
next_material_7_ID := next_material_information[6].ID;
next_material_7_QTY := next_material_information[6].QTY;
next_material_8_ID := next_material_information[7].ID;
next_material_8_QTY := next_material_information[7].QTY;
next_material_9_ID := next_material_information[8].ID;
next_material_9_QTY := next_material_information[8].QTY;
next_material_10_ID := next_material_information[9].ID;
next_material_10_QTY := next_material_information[9].QTY;
next_material_11_ID := next_material_information[10].ID;
next_material_11_QTY := next_material_information[10].QTY;
next_material_12_ID := next_material_information[11].ID;
next_material_12_QTY := next_material_information[11].QTY;
next_material_13_ID := next_material_information[12].ID;
next_material_13_QTY := next_material_information[12].QTY;
next_material_14_ID := next_material_information[13].ID;
next_material_14_QTY := next_material_information[13].QTY;
next_material_15_ID := next_material_information[14].ID;
next_material_15_QTY := next_material_information[14].QTY;

mark_BUBD := mark_bubd_information.BestUsedByDate;
mark_prefix := mark_bubd_information.Prefix;
mark_format := mark_bubd_information.Format;

IF	csp_main_phaseManager.p_mes_interface_enable
THEN
	IF	csp_main.i_start_job_request
	THEN
		led_set_status(
			status				:= HMI_OBJECT_STATUS_ON, 
			CONVERSION_this		:= order_valid_led);
			
		led_set_status(
			status				:= HMI_OBJECT_STATUS_ON, 
			CONVERSION_this		:= product_valid_led);

		led_set_status(
			status				:= HMI_OBJECT_STATUS_ON, 
			CONVERSION_this		:= recipe_valid_led);

		led_set_status(
			status				:= HMI_OBJECT_STATUS_ON, 
			CONVERSION_this		:= materials_valid_led);

		led_set_status(
			status				:= HMI_OBJECT_STATUS_ON, 
			CONVERSION_this		:= mark_valid_led);		
	
		IF	csp_main.i_csp_data_ref^.Status.Job.4
			OR
			csp_main.i_csp_data_ref^.Status.Job.5
		THEN
			led_set_color(
				color				:= HMI_LED_COLOR_RED, 
				CONVERSION_this		:= order_valid_led);
		ELSE
			led_set_color(
				color				:= HMI_LED_COLOR_GREEN, 
				CONVERSION_this		:= order_valid_led);			
		END_IF	
		
		IF	csp_main.i_csp_data_ref^.Status.Job.6
			OR
			csp_main.i_csp_data_ref^.Status.Job.7
		THEN
			led_set_color(
				color				:= HMI_LED_COLOR_RED, 
				CONVERSION_this		:= product_valid_led);
		ELSE
			led_set_color(
				color				:= HMI_LED_COLOR_GREEN, 
				CONVERSION_this		:= product_valid_led);			
		END_IF	

		IF	csp_main.i_csp_data_ref^.Status.Job.8
			OR
			csp_main.i_csp_data_ref^.Status.Job.9
		THEN
			led_set_color(
				color				:= HMI_LED_COLOR_RED, 
				CONVERSION_this		:= recipe_valid_led);
		ELSE
			led_set_color(
				color				:= HMI_LED_COLOR_GREEN, 
				CONVERSION_this		:= recipe_valid_led);			
		END_IF	

		IF	csp_main.i_csp_data_ref^.Status.Job.10
			OR
			csp_main.i_csp_data_ref^.Status.Job.11
		THEN
			led_set_color(
				color				:= HMI_LED_COLOR_RED, 
				CONVERSION_this		:= materials_valid_led);
		ELSE
			led_set_color(
				color				:= HMI_LED_COLOR_GREEN, 
				CONVERSION_this		:= materials_valid_led);			
		END_IF	

		IF	csp_main.i_csp_data_ref^.Status.Job.12
			OR
			csp_main.i_csp_data_ref^.Status.Job.13
		THEN
			led_set_color(
				color				:= HMI_LED_COLOR_RED, 
				CONVERSION_this		:= mark_valid_led);
		ELSE
			led_set_color(
				color				:= HMI_LED_COLOR_GREEN, 
				CONVERSION_this		:= mark_valid_led);			
		END_IF			
	END_IF
ELSE
		led_set_status(
			status				:= HMI_OBJECT_STATUS_OFF, 
			CONVERSION_this		:= order_valid_led);
			
		led_set_status(
			status				:= HMI_OBJECT_STATUS_OFF, 
			CONVERSION_this		:= product_valid_led);

		led_set_status(
			status				:= HMI_OBJECT_STATUS_OFF, 
			CONVERSION_this		:= recipe_valid_led);

		led_set_status(
			status				:= HMI_OBJECT_STATUS_OFF, 
			CONVERSION_this		:= materials_valid_led);

		led_set_status(
			status				:= HMI_OBJECT_STATUS_OFF, 
			CONVERSION_this		:= mark_valid_led);		
END_IF
END_ACTION

ACTION run_cycle:
IF	csp_main_phaseManager.fsm_status <> CSP_MAIN_PHASE_MANAGER_STATUS_START_JOB_10
THEN	
	fsm_status := 0;
END_IF

fsm_enable_conditions :=
	(
		csp_main_phaseManager.fsm_status
		=
		CSP_MAIN_PHASE_MANAGER_STATUS_START_JOB_10
	);
	
IF	(
			(
				NOT fsm_enable_conditions
				OR
				(
					NOT csp_main.i_start_job_request
					AND
					NOT csp_main.i_cycle_enable_request
				)
			)
		AND
		(start_job_running
		OR
		next_material_information[csp_main_phaseManager.MASTER_CASE_BLANK_MATERIAL_ID].ID = 'None') // 'None' is set when running club LCNC, resets Status_Job to a value of 1 (unscheduled)
	)
THEN
	fsm_status := 666;
END_IF

CASE fsm_status OF
	0:

		//csp_main.i_csp_data_ref^.Status.Job := 1;		(* Not Scheduled *)	
	
		check_order_information := FALSE;
		check_product_information := FALSE;
		check_recipe_information := FALSE;
		check_curr_material_information := FALSE;
		check_next_material_information := FALSE;
		check_mark_bubd_information := FALSE;
	
		check_MES_variables := FALSE;
	
		IF fsm_enable_conditions
		THEN
			fsm_status := 10;
		END_IF
		
	10:

		IF csp_main.i_start_job_request
		THEN
			start_job_running := TRUE;
			i_end_job_done^ := FALSE;			
			//csp_main.i_csp_data_ref^.Status.Job := 2;		(* Job is In Progress *)					
			fsm_status := 20;
		END_IF
		
	15:
		// Reset mark,current_material,order,product information before get a new job
		csp_main.i_mark_bubd_information^.BestUsedByDate 	:= '';
		csp_main.i_mark_bubd_information^.Prefix 			:= '';
		csp_main.i_mark_information^.ID 					:= '';
		csp_main.i_mark_information^.KdpSite 				:= '';
		csp_main.i_mark_information^.OriginDate 			:= '';
		csp_main.i_mark_information^.PartnerSite			:= '';
		csp_main.i_mark_information^.Template.Carton		:= '';
		csp_main.i_mark_information^.Template.CASEPACK		:= '';
		csp_main.i_mark_information^.Template.Pod			:= '';
		//csp_main.i_mark_kdp_site_information^				:= '';
		
		csp_main.i_current_material_information^[0].ID 		:= '';
		csp_main.i_current_material_information^[0].QTY		:= 0;
		csp_main.i_next_material_information^[0].ID			:= '';
		csp_main.i_next_material_information^[0].QTY		:= 0;

		csp_main.i_current_material_information^[1].ID 		:= '';
		csp_main.i_current_material_information^[1].QTY		:= 0;
		csp_main.i_next_material_information^[1].ID			:= '';
		csp_main.i_next_material_information^[1].QTY		:= 0;

		csp_main.i_current_material_information^[2].ID 		:= '';
		csp_main.i_current_material_information^[2].QTY		:= 0;
		csp_main.i_next_material_information^[2].ID			:= '';
		csp_main.i_next_material_information^[2].QTY		:= 0;

		csp_main.i_current_material_information^[3].ID 		:= '';
		csp_main.i_current_material_information^[3].QTY		:= 0;
		csp_main.i_next_material_information^[3].ID			:= '';
		csp_main.i_next_material_information^[3].QTY		:= 0;

		csp_main.i_current_material_information^[4].ID 		:= '';
		csp_main.i_current_material_information^[4].QTY		:= 0;
		csp_main.i_next_material_information^[4].ID			:= '';
		csp_main.i_next_material_information^[4].QTY		:= 0;
        
		csp_main.i_recipe_information^.Cartoner				:= '';	
		csp_main.i_next_recipe_information^.Cartoner		:= '';
		csp_main.i_recipe_information^.Filler				:= '';
		csp_main.i_next_recipe_information^.Filler			:= '';					
		csp_main.i_recipe_information^.CasePacker			:= '';
		csp_main.i_next_recipe_information^.CasePacker		:= '';	
        
		csp_main.i_order_information^.ID					:= '';	
		csp_main.i_order_information^.SapBatchID			:= '';
		csp_main.i_product_information^.CaffeinatedFlag		:= FALSE;
		csp_main.i_product_information^.CartonsPerCase		:= 0;
		csp_main.i_product_information^.FillWeight.Maximum	:= 0;
		csp_main.i_product_information^.FillWeight.Minimum	:= 0;
		csp_main.i_product_information^.FillWeight.Target	:= 0;
		csp_main.i_product_information^.FilterType			:= '';
		csp_main.i_product_information^.FlavorDose			:= 0;
		csp_main.i_product_information^.FlavorFlag			:= FALSE;
		csp_main.i_product_information^.ID					:= '';
		csp_main.i_product_information^.UPC					:= '';
		csp_main.i_product_information^.KosherFlag			:= FALSE;
		csp_main.i_product_information^.OrganicFlag			:= FALSE;
		csp_main.i_product_information^.PodsPerCarton		:= 0;
		csp_main.i_product_information^.PodsPerCase			:= 0;
		csp_main.i_product_information^.ShelfLife			:= 0;
		csp_main.i_next_order_information^.ID						:= '';	
		csp_main.i_next_order_information^.SapBatchID				:= '';
		csp_main.i_next_product_information^.CaffeinatedFlag		:= FALSE;
		csp_main.i_next_product_information^.CartonsPerCase			:= 0;
		csp_main.i_next_product_information^.FillWeight.Maximum		:= 0;
		csp_main.i_next_product_information^.FillWeight.Minimum		:= 0;
		csp_main.i_next_product_information^.FillWeight.Target		:= 0;
		csp_main.i_next_product_information^.FilterType				:= '';
		csp_main.i_next_product_information^.FlavorDose				:= 0;
		csp_main.i_next_product_information^.FlavorFlag				:= FALSE;
		csp_main.i_next_product_information^.ID						:= '';
		csp_main.i_next_product_information^.UPC					:= '';
		csp_main.i_next_product_information^.KosherFlag				:= FALSE;
		csp_main.i_next_product_information^.OrganicFlag			:= FALSE;
		csp_main.i_next_product_information^.PodsPerCarton			:= 0;
		csp_main.i_next_product_information^.PodsPerCase			:= 0;
		csp_main.i_next_product_information^.ShelfLife				:= 0;	
	
		fsm_status := 20;				
		
	20:
		order_information := csp_main.i_order_information^;
		product_information := csp_main.i_product_information^;
		recipe_information := csp_main.i_recipe_information^;
		current_material_information := csp_main.i_current_material_information^;
		next_material_information := csp_main.i_next_material_information^;
		mark_bubd_information := csp_main.i_mark_bubd_information^;
		
		fsm_status := 30;
		
	30:
		check_MES_variables := TRUE;
		fsm_status := 40;

	40:
		IF MES_variables_valid
		THEN
		
			check_MES_variables := FALSE;
			fsm_status := 110;
			csp_main.i_csp_data_ref^.Status.Job := 2;
		ELSE
			csp_main.i_csp_data_ref^.Status.Job.5 := NOT order_valid;
			csp_main.i_csp_data_ref^.Status.Job.7 := NOT product_valid;
			csp_main.i_csp_data_ref^.Status.Job.9 := NOT recipe_valid;
			//csp_main.i_csp_data_ref^.Status.Job.11 := (NOT curr_material_valid OR NOT next_material_valid);
			csp_main.i_csp_data_ref^.Status.Job.11 := NOT curr_material_valid;
			csp_main.i_csp_data_ref^.Status.Job.13 := NOT mark_bubd_valid;
			
			fsm_status := 666;
		END_IF
	

	110:
		IF 	csp_main.i_cycle_enable_request
			AND 
			NOT csp_main.i_start_job_request
		THEN
			fsm_status := 555;
		(*ELSIF	(NOT boolean_or_get_status(machine_setup_completed_bor))
		THEN
			execute_machine_setup := TRUE;
			fsm_status := 100;*)
		END_IF
		
	555:
		start_job_running := FALSE;
		start_job_done := TRUE;
		
		IF	NOT csp_main.i_cycle_enable_request
		THEN
			start_job_running := FALSE;
			start_job_done := FALSE;

			fsm_status := 0;
		END_IF
		
	666:
		start_job_running := FALSE;
		start_job_done := FALSE;
		
		IF NOT csp_main.i_start_job_request
		THEN
			fsm_status := 0;
		ELSE
			IF NOT MES_variables_valid
			THEN
				fsm_status := 20;
			END_IF
		END_IF
END_CASE
END_ACTION

END_PROGRAM

// ---- Application/CSP/Main/Phase Manager/csp_main_phaseManager.TcPOU
(*********************************** G.D S.p.A. - Technical Department ***********************************
============= PROGRAM INFO ============
FOLDER:             TBD
MACHINES INVOLVED:  TBD 

============= DESCRIPTION =============
WN phase manager program

============= REVISIONS ===============
Date		Version	 	Author      	Description             
----------	-------		------------  	--------------------------------------------
2020/06/16 	0000.00	 	G.Cera 			Creation of the PRG
2021/04/09 	0000.01	 	M.Grasso	 	Flow Chart version
**********************************************************************************************************)
(*$R
	process_ref := prc;
$*)
PROGRAM csp_main_phaseManager
VAR
	prc:												process;
	prc_path:											STRING;																		

	start_MES_variables_update:							BOOL;
	
	start_job_completed:								BOOL;
	//steady_state_completed:								BOOL;
	//cup_supply_completed:								BOOL;
	//carton_case_supply_completed:						BOOL;
	//production_completed:								BOOL;
	//near_end_of_run_completed:						BOOL;
	runout_completed:									BOOL;
		
	(*TOTAL RUNNING TIME additional variables*)
	mch_running_tmr:									timer;
	refresh_tmr:										timer;

	mch_running_rtrig:									R_TRIG;
	
	mch_running_elapsed_time_nvr:						LREAL;
	mch_running_elapsed_time_mem_nvr:					LREAL;
	timer_to_be_removed:								LREAL;

	mch_order_tmr:										timer;
	(*****)
	
	start_job_green_label:								hmi_graphic_object_status;
	steady_state_green_label:							hmi_graphic_object_status;
	cups_supply_green_label:							hmi_graphic_object_status;
	carton_cases_supply_green_label:					hmi_graphic_object_status;
	production_green_label:								hmi_graphic_object_status;
	completion_green_label:								hmi_graphic_object_status;
	runout_green_label:									hmi_graphic_object_status;
	end_job_green_label:								hmi_graphic_object_status;
	
	mes_interface_enable_prow:							parameter_overwrite;
	mes_interface_enable_old:							BOOL;
	
	mes_interface_disabled_wsm:							message;
	mes_alarm_start_job_asm:							csp_main_phMan_start_job_snapshot;
	mes_alarm_asm:										csp_main_phaseManager_snapshot;
	mes_warning_wsm:									csp_main_phaseManager_warning_snapshot;
	mes_alarm_string:									STRING;
	mes_warning_string:									STRING;	
	
	change_order_ID:									BOOL;
	
	(* MES production variables *)
	//Status variables
	current_job_status:									DINT;								(*$M $*)
	next_job_status:									DINT;								(*$M $*)
	filler_ready_for_coffee:							BOOL;								(*$M $*)	
	machine_running:									BOOL;								(*$M $*)
	filler_faulted:										BOOL;								(*$M $*)
	cup_automation_faulted:								BOOL;								(*$M $*)
	disk_automation_faulted:							BOOL;								(*$M $*)	
	filter_automation_faulted:							BOOL;								(*$M $*)	
	lid_automation_faulted:								BOOL;								(*$M $*)	
	run_out_in_progress:								BOOL;								(*$M $*)
	run_out_completed:									BOOL;								(*$M $*)
	target_speed_cupspmin:								INT;								(*$M unit := cups/min; $*)
	actual_speed_cupspmin:								INT;								(*$M unit := cups/min; $*)
	actual_speed_poundspmin:							INT;								(*$M unit := pounds/min; $*)
	current_stop_reason:								DINT;								(*$M $*)
	emergency_stop_active:								BOOL;								(*$M $*)
	guard_open_stop_active:								BOOL;								(*$M $*)
	operator_stop_active:								BOOL;								(*$M $*)
	infeed_cups_missing:								BOOL;								(*$M $*)
	infeed_filters_missing:								BOOL;								(*$M $*)
	infeed_disks_missing:								BOOL;								(*$M $*)
	infeed_coffee_missing:								BOOL;								(*$M $*)
	infeed_lids_missing:								BOOL;								(*$M $*)	
	downstream_block:									BOOL;								(*$M $*)
	reject_block:										BOOL;								(*$M $*)
	waste_block:										BOOL;								(*$M $*)

	//Start variables
	csp_start_request:									BOOL;								(*$M $*)	
	csp_start_ramp:										BOOL;								(*$M $*)
	csp_start_peak_wait:								BOOL;								(*$M $*)	
	
	//Production variables
	current_order_started_pods:							DINT;								(*$M unit := cups; $*)
	current_order_good_pods:							DINT;								(*$M unit := cups; $*)
	total_started_cups:									DINT;								(*$M unit := cups; $*)
	total_good_cups:									DINT;								(*$M unit := cups; $*)
	total_reject_cups:									DINT;								(*$M unit := cups; $*)
	current_order_time_min:								DINT;								(*$M unit := min; $*)
	current_order_running_time_min:						DINT;								(*$M unit := min; $*)
	rejected_cups_percentage:							DINT;								(*$M unit := %; $*)
	calculated_cups_with_remaining_coffee:				DINT;								(*$M unit := cups; $*)	
	current_order_no_cup_rejects:						DINT;								(*$M unit := cups; $*)	
	current_order_no_disk_rejects:						DINT;								(*$M unit := cups; $*)	
	current_order_no_filter_rejects:			    	DINT;								(*$M unit := cups; $*)	
	current_order_over_weight_rejects:					DINT;								(*$M unit := cups; $*)	
	current_order_under_weight_rejects:					DINT;								(*$M unit := cups; $*)	
	current_order_no_lid_rejects:						DINT;								(*$M unit := cups; $*)	
	current_order_leak_test_rejects:					DINT;								(*$M unit := cups; $*)	
	current_order_bad_filter_rejects:					DINT;								(*$M unit := cups; $*)	
	current_order_sample_rejects:						DINT;								(*$M unit := cups; $*)	
	current_order_consumed_cups:						DINT;								(*$M unit := cups; $*)
	current_order_consumed_disks:						DINT;								(*$M unit := disks; $*)
	current_order_consumed_filters:						DINT;								(*$M unit := filters; $*)
	current_order_consumed_coffee:						REAL;								(*$M unit := pounds; $*)
	current_order_consumed_flavor:						REAL;								(*$M unit := ml; $*)
	current_order_consumed_lids:						DINT;								(*$M unit := lids; $*)

	
	//CT calls variables
	ctCall_low_cup_supply:								BOOL;								(*$M $*)
	ctCall_low_disk_supply:								BOOL;								(*$M $*)
	ctCall_low_lid_supply:								BOOL;								(*$M $*)
	ctCall_low_filter_supply:							BOOL;								(*$M $*)
	ctCall_scrap_full:									BOOL;								(*$M $*)
	ctCall_main_fault:									BOOL;								(*$M $*)
	ctCall_cup_automation_fault:						BOOL;								(*$M $*)
	ctCall_disk_automation_fault:						BOOL;								(*$M $*)
	ctCall_lid_automation_fault:						BOOL;								(*$M $*)
	ctCall_filter_automation_fault:						BOOL;								(*$M $*)


	//Take Away system variables	
	foil_and_paper_take_away_system_run_request:		BOOL;								(*$M $*)
	foil_and_paper_take_away_system_run_status:			BOOL;								(*$M $*)
	stop_from_foil_and_paper_take_away_system:			BOOL;								(*$M $*)
	foil_and_paper_take_away_system_faulted_status:		BOOL;								(*$M $*)
	

	//Dock variables
	dock_1_drop_available:								BOOL;								(*$M $*)
	dock_1_pick_available:								BOOL;								(*$M $*)
	dock_1_AMR_ready_to_receive:						BOOL;								(*$M $*)						
	dock_1_pick_location_conveyor_energized:			BOOL;								(*$M $*)
	dock_1_AMR_conveyor_top_fault_code:					DINT;								(*$M $*)
	dock_2_drop_available:								BOOL;								(*$M $*)
	dock_2_pick_available:								BOOL;								(*$M $*)
	dock_2_AMR_ready_to_receive:						BOOL;								(*$M $*)						
	dock_2_pick_location_conveyor_energized:			BOOL;								(*$M $*)
	dock_2_AMR_conveyor_top_fault_code:					DINT;								(*$M $*)


	//Coffe supply system variables


	upstream_coffee_no_active_job:						BOOL;								(*$M $*)
	upstream_coffee_supplying_coffee:					BOOL;								(*$M $*)
	upstream_coffee_order_complete_tubo_empty:			BOOL;								(*$M $*)
	upstream_coffee_faulted:							BOOL;								(*$M $*)
	upstream_coffee_silo_low:							BOOL;								(*$M $*)
	upstream_coffee_tube_high:							BOOL;								(*$M $*)
	upstream_coffee_tube_med:							BOOL;								(*$M $*)
	upstream_coffee_tube_low:							BOOL;								(*$M $*)
	


	machine_running_led:								led;	
	filler_faulted_led:									led;	
	ready_for_coffee_led:								led;	
	cup_automation_faulted_led:							led;	
	disk_automation_faulted_led:						led;
	filter_automation_faulted_led:						led;
	lid_automation_faulted_led:							led;	
	runout_in_progress_led:								led;	
	runout_completed_led:								led;	
	estop_active_led:									led;	
	guard_open_led:										led;	
	operator_stop_led:									led;	
	infeed_cups_missing_led:							led;				
	infeed_filters_missing_led:							led;				
	infeed_disks_missing_led:							led;			
	infeed_coffee_missing_led:							led;		
	infeed_lids_missing_led:							led;
	downstream_block_led:								led;
	reject_block_led:									led;
	waste_block_led:									led;	
	filler_start_request_led:							led;	
	filler_start_ramp_led:								led;
	filler_start_peak_wait_led:							led;
	dock_1_drop_available_led:							led;
	dock_1_pick_available_led:							led;
	dock_1_AMR_ready_to_receive_led:					led;						
	dock_1_pick_location_conveyor_energized_led:		led;
	dock_2_drop_available_led:							led;
	dock_2_pick_available_led:							led;
	dock_2_AMR_ready_to_receive_led:					led;						
	dock_2_pick_location_conveyor_energized_led:		led;
	dock_2_AMR_conveyor_top_fault_code_led:				led;
	ctCall_low_cup_supply_led:							led;
	ctCall_low_disk_supply_led:							led;
	ctCall_low_lid_supply_led:							led;
	ctCall_low_filter_supply_led:						led;
	ctCall_scrap_full_led:								led;
	ctCall_main_fault_led:								led;
	ctCall_cup_automation_fault_led:					led;
	ctCall_disk_automation_fault_led:					led;
	ctCall_lid_automation_fault_led:					led;
	ctCall_filter_automation_fault_led:					led;
	
	
	p_mes_interface_enable:								BOOL; 	(*$P desc := if TRUE, phase manager transitions are commanded by MES system; $*)
	p_last_case:										BOOL;	(*$P $*)
	confirm_run_out_mode_pow:							parameter_overwrite;
	first_cycle:										BOOL;	//this bit prevents the phase manager cycle to restart when the machine is switched on			

	
	
	TEST_BOOL:											BOOL;
	TEST_DINT:											DINT;
	
	bt_1sec:											TON;
	bt_1sec_aux:										BOOL;
	i_start_job_done:									POINTER TO BOOL;
	stop_message_CSP_ref:								POINTER TO message;
	
END_VAR

VAR PERSISTENT
	fsm_status:											csp_main_phaseManager_status_enum;		(*$M desc := phase manager status; $*)														
	mes_elapsed_time_1_npr:								UDINT;	(*$M desc := Time1; $*)	
	mes_elapsed_time_2_npr:								UDINT; 	(*$M desc := Time2; $*)
END_VAR

VAR CONSTANT
	MASTER_CASE_BLANK_MATERIAL_ID:						INT:=6;
	CASE_LABEL_MATERIAL_ID:								INT:=7;
END_VAR

_read_var_input();

_object_manager();

IF NOT objects_running()
THEN
	RETURN;	
END_IF

_read_process_image();

_mode_manager();

CASE process_get_mode(prc) of
	MODE_ABSENT,
	MODE_INACTIVE:
		RETURN;
	MODE_TEST:
		_handle_process_test();
END_CASE

_set_runtime_properties();

(********************************* BODY *********************************)

IF first_cycle
THEN	
	mes_interface_enable_old := TRUE;
	IF p_mes_interface_enable
	THEN
		first_cycle := FALSE;
	ELSE
		parameter_overwrite_set_bool_value(
			value				:= TRUE, 
			CONVERSION_this		:= mes_interface_enable_prow);	
	END_IF
END_IF;	

IF	(
		mes_interface_enable_old
		<>
		p_mes_interface_enable
	)
	AND
	NOT first_cycle
THEN
	IF machine_is_stopped(csp.mch)
	THEN
		mes_interface_enable_old := p_mes_interface_enable;
	ELSE
		parameter_overwrite_set_bool_value(
			value				:= mes_interface_enable_old, 
			CONVERSION_this		:= mes_interface_enable_prow);
	END_IF
END_IF

csp_main.i_csp_data_ref^.Status.Online	:=	p_mes_interface_enable;

(************************************************************************)

start_job_completed		:=	csp_main_phaseManager_startJob.start_job_done;
runout_completed		:=	csp_main_phaseManager_run_out.run_out_done;

IF csp_main.i_csp_data_ref^.Status.RunOutComplete AND NOT p_last_case
THEN
	parameter_overwrite_set_bool_value(TRUE, confirm_run_out_mode_pow);
END_IF

(**************************** PROGRAM HANDLER ***************************)
run_cycle();
custom_page();
variables_update();
(************************************************************************)

_handle_messages();

_write_output();

ACTION _handle_messages:
IF	p_mes_interface_enable
THEN
	process_message_reset(mes_interface_disabled_wsm);
	
	IF	csp_customerInterfaces.MES.Alarm <> 0
	THEN		

		CASE csp_customerInterfaces.MES.Alarm OF
			1:	mes_alarm_string := 'JOB NOT SCHEDULED';	
			2:	mes_alarm_string := 'JOB PENDING';
			
			ELSE mes_alarm_string := 'ALARM CODE NON DEFINED';
			
		END_CASE	
	
		csp_main_phaseManager_set_snapshot(
			errorID_1			:= csp_customerInterfaces.MES.Alarm, 
			errorID_2			:= 0, 
			errorID_3			:= 0, 
			reason				:= mes_alarm_string, 
			job_not_scheduled	:= csp_customerInterfaces.MES.Alarm.0, 
			job_pending			:=csp_customerInterfaces.MES.Alarm.1, 
			CONVERSION_this		:= mes_alarm_asm);
	ELSE
		process_message_reset(mes_alarm_asm.message);			
	END_IF		

	IF	csp_customerInterfaces.MES.Warning <> 0
	THEN		

		CASE csp_customerInterfaces.MES.Warning OF
			1:	mes_warning_string := 'MAINTENANCE JOB ACTIVE';	
						
			ELSE mes_warning_string := 'WARNING CODE NON DEFINED';
			
		END_CASE	
	
		csp_main_phaseManager_warning_set_snapshot(
			errorID_1				:= csp_customerInterfaces.MES.Warning, 
			errorID_2				:= 0, 
			errorID_3				:= 0, 
			reason					:= mes_warning_string, 
			maintenance_job_active	:= csp_customerInterfaces.MES.Warning.0, 
			CONVERSION_this			:= mes_warning_wsm);
	ELSE
		process_message_reset(mes_warning_wsm.message);			
	END_IF
	
ELSE
	process_message_set(
		errorID_1			:= 1, 
		errorID_2			:= 0, 
		errorID_3			:= 0, 
		CONVERSION_this		:= mes_interface_disabled_wsm);
		
	process_message_reset(mes_alarm_asm.message);	
	process_message_reset(mes_warning_wsm.message);	
END_IF

IF	(
		csp_main_phaseManager_startJob.fsm_status
		=
		666
	)
THEN
	csp_main_phMan_start_job_set_snapshot(
		errorID_1			:= fsm_status, 
		errorID_2			:= csp_main.i_csp_data_ref^.Status.Job, 
		errorID_3			:= 0, 
		reason				:= 'MES INCORRECT INFORMATION', 
		order_valid			:= csp_main_phaseManager_startJob.order_valid, 
		product_valid		:= csp_main_phaseManager_startJob.product_valid, 
		recipe_valid		:= csp_main_phaseManager_startJob.recipe_valid, 
		materials_valid		:= (csp_main_phaseManager_startJob.curr_material_valid AND csp_main_phaseManager_startJob.next_material_valid), 
		mark_valid			:= csp_main_phaseManager_startJob.mark_bubd_valid, 
		CONVERSION_this		:= mes_alarm_start_job_asm);
ELSE
	process_message_reset(mes_alarm_start_job_asm.message);
END_IF
END_ACTION

ACTION _handle_process_test:
;
END_ACTION

ACTION _mode_manager:
IF process_mode_req_is_pending(prc)
THEN
    process_apply_mode_req_first_step(prc);
    CASE process_get_mode(prc) OF
        MODE_TO_ABSENT:
			;
        MODE_TO_INACTIVE:
			;
        MODE_TO_TEST:
			;
        MODE_TO_OPERATIONAL:
			;
    END_CASE
    process_apply_mode_req_second_step(prc);
END_IF
END_ACTION

ACTION _object_manager:
IF objects_initialization()
THEN
	sub_process_init(
		object_name					:= 'csp_main_phaseManager.prc', 
		process						:= csp_main.prc, 
		CONVERSION_this				:= prc);
		
	prc_path 						:= process_get_path(prc);
	
	parameter_overwrite_bool_init(
		object_name					:= CONCAT(prc_path, '_mes_interface_enable_prow'), 
		parameter					:= p_mes_interface_enable, 
		process						:= prc, 
		CONVERSION_this				:= mes_interface_enable_prow);
		
	timer_init(
		object_name					:=	CONCAT(prc_path, '_mch_running_tmr'),
		process						:=	prc,
		CONVERSION_this				:=	mch_running_tmr);
		
	timer_init(
		object_name					:=	CONCAT(prc_path, '_refresh_tmr'),
		process						:=	prc,
		CONVERSION_this				:=	refresh_tmr);
		
	timer_init(
		object_name					:=	CONCAT(prc_path, '_mch_order_tmr'),
		process						:=	prc,
		CONVERSION_this				:=	mch_order_tmr);	
		
	process_message_init(
		object_name					:= CONCAT(prc_path, '_mes_interface_disabled_wsm'), 
		behaviour					:= MESSAGE_BEHAVIOUR_STATE, 
		reset_timeout				:= 0, 
		disableable					:= FALSE, 
		individual_reset			:= FALSE, 
		machine_reaction			:= MACHINE_REACTION_NO_STOP, 
		typology					:= MESSAGE_TYPOLOGY_NORMAL, 
		process						:= prc, 
		CONVERSION_this				:= mes_interface_disabled_wsm);
		
	csp_main_phMan_start_job_init_snapshot(
		message_name				:= CONCAT(prc_path, '_mes_alarm_start_job_asm'), 
		behaviour					:= MESSAGE_BEHAVIOUR_TRY_AND_CHECK, 
		reset_timeout				:= 500, 
		disableable					:= FALSE, 
		individual_reset			:= FALSE, 
		machine_reaction			:= MACHINE_REACTION_NORMAL_STOP, 
		typology					:= MESSAGE_TYPOLOGY_ABNORMAL, 
		process						:= prc, 
		CONVERSION_this				:= mes_alarm_start_job_asm);			
		
	csp_main_phaseManager_init_snapshot(
		message_name				:= CONCAT(prc_path, '_mes_alarm_asm'), 
		behaviour					:= MESSAGE_BEHAVIOUR_STATE, 
		reset_timeout				:= 0, 
		disableable					:= FALSE, 
		individual_reset			:= FALSE, 
		machine_reaction			:= MACHINE_REACTION_NORMAL_STOP, 
		typology					:= MESSAGE_TYPOLOGY_ABNORMAL, 
		process						:= prc, 
		CONVERSION_this				:= mes_alarm_asm);	

	csp_main_phaseManager_warning_init_snapshot(
		message_name				:= CONCAT(prc_path, '_mes_warning_wsm'), 
		behaviour					:= MESSAGE_BEHAVIOUR_STATE, 
		reset_timeout				:= 0, 
		disableable					:= FALSE, 
		individual_reset			:= FALSE, 
		machine_reaction			:= MACHINE_REACTION_NO_STOP, 
		typology					:= MESSAGE_TYPOLOGY_NORMAL, 
		process						:= prc, 
		CONVERSION_this				:= mes_warning_wsm);	
		
	hmi_graphic_object_status_init(
		object_name					:= CONCAT(prc_path, '_start_job_green_label'), 
		process						:= prc, 
		CONVERSION_this				:= start_job_green_label);
		
	hmi_graphic_object_status_init(
		object_name					:= CONCAT(prc_path, '_steady_state_green_label'), 
		process						:= prc, 
		CONVERSION_this				:= steady_state_green_label);

	hmi_graphic_object_status_init(
		object_name					:= CONCAT(prc_path, '_cups_supply_green_label'), 
		process						:= prc, 
		CONVERSION_this				:= cups_supply_green_label);

	hmi_graphic_object_status_init(
		object_name					:= CONCAT(prc_path, '_carton_cases_supply_green_label'), 
		process						:= prc, 
		CONVERSION_this				:= carton_cases_supply_green_label);

	hmi_graphic_object_status_init(
		object_name					:= CONCAT(prc_path, '_production_green_label'), 
		process						:= prc, 
		CONVERSION_this				:= production_green_label);

	hmi_graphic_object_status_init(
		object_name					:= CONCAT(prc_path, '_completion_green_label'), 
		process						:= prc, 
		CONVERSION_this				:= completion_green_label);

	hmi_graphic_object_status_init(
		object_name					:= CONCAT(prc_path, '_runout_green_label'), 
		process						:= prc, 
		CONVERSION_this				:= runout_green_label);	

	hmi_graphic_object_status_init(
		object_name					:= CONCAT(prc_path, '_end_job_green_label'), 
		process						:= prc, 
		CONVERSION_this				:= end_job_green_label);

	led_init(
		object_name					:= CONCAT(prc_path, '_machine_running_led'), 
		process						:= prc, 
		CONVERSION_this				:= machine_running_led);	
		
	led_init(
		object_name					:= CONCAT(prc_path, '_filler_faulted_led'), 
		process						:= prc, 
		CONVERSION_this				:= filler_faulted_led);

	led_init(
		object_name					:= CONCAT(prc_path, '_ready_for_coffee_led'), 
		process						:= prc, 
		CONVERSION_this				:= ready_for_coffee_led);		

	led_init(
		object_name					:= CONCAT(prc_path, '_cup_automation_faulted_led'), 
		process						:= prc, 
		CONVERSION_this				:= cup_automation_faulted_led);
		
	led_init(
		object_name					:= CONCAT(prc_path, '_disk_automation_faulted_led'), 
		process						:= prc, 
		CONVERSION_this				:= disk_automation_faulted_led);		
		
	led_init(
		object_name					:= CONCAT(prc_path, '_filter_automation_faulted_led'), 
		process						:= prc, 
		CONVERSION_this				:= filter_automation_faulted_led);		

	led_init(
		object_name					:= CONCAT(prc_path, '_lid_automation_faulted_led'), 
		process						:= prc, 
		CONVERSION_this				:= lid_automation_faulted_led);		

	led_init(
		object_name					:= CONCAT(prc_path, '_runout_in_progress_led'), 
		process						:= prc, 
		CONVERSION_this				:= runout_in_progress_led);

	led_init(
		object_name					:= CONCAT(prc_path, '_runout_completed_led'), 
		process						:= prc, 
		CONVERSION_this				:= runout_completed_led);	

	led_init(
		object_name					:= CONCAT(prc_path, '_estop_active_led'), 
		process						:= prc, 
		CONVERSION_this				:= estop_active_led);	
		
	led_init(
		object_name					:= CONCAT(prc_path, '_guard_open_led'), 
		process						:= prc, 
		CONVERSION_this				:= guard_open_led);

	led_init(
		object_name					:= CONCAT(prc_path, '_operatpr_stop_led'), 
		process						:= prc, 
		CONVERSION_this				:= operator_stop_led);
		
	led_init(
		object_name					:= CONCAT(prc_path, '_infeed_cups_missing_led'), 
		process						:= prc, 
		CONVERSION_this				:= infeed_cups_missing_led);

	led_init(
		object_name					:= CONCAT(prc_path, '_infeed_filters_missing_led'), 
		process						:= prc, 
		CONVERSION_this				:= infeed_filters_missing_led);

	led_init(
		object_name					:= CONCAT(prc_path, '_infeed_disks_missing_led'), 
		process						:= prc, 
		CONVERSION_this				:= infeed_disks_missing_led);

	led_init(
		object_name					:= CONCAT(prc_path, '_infeed_coffee_missing_led'), 
		process						:= prc, 
		CONVERSION_this				:= infeed_coffee_missing_led);

	led_init(
		object_name					:= CONCAT(prc_path, '_infeed_lids_missing_led'), 
		process						:= prc, 
		CONVERSION_this				:= infeed_lids_missing_led);		
		
	led_init(
		object_name					:= CONCAT(prc_path, '_downstream_block_led'), 
		process						:= prc, 
		CONVERSION_this				:= downstream_block_led);

	led_init(
		object_name					:= CONCAT(prc_path, '_reject_block_led'), 
		process						:= prc, 
		CONVERSION_this				:= reject_block_led);

	led_init(
		object_name					:= CONCAT(prc_path, '_waste_block_led'), 
		process						:= prc, 
		CONVERSION_this				:= waste_block_led);		
		
	led_init(
		object_name					:= CONCAT(prc_path, '_filler_start_request_led'), 
		process						:= prc, 
		CONVERSION_this				:= filler_start_request_led);

	led_init(
		object_name					:= CONCAT(prc_path, '_filler_start_ramp_led'), 
		process						:= prc, 
		CONVERSION_this				:= filler_start_ramp_led);

	led_init(
		object_name					:= CONCAT(prc_path, '_filler_start_peak_wait_led'), 
		process						:= prc, 
		CONVERSION_this				:= filler_start_peak_wait_led);		

	led_init(
		object_name					:= CONCAT(prc_path, '_dock_1_drop_available_led'), 
		process						:= prc, 
		CONVERSION_this				:= dock_1_drop_available_led);	

	led_init(
		object_name					:= CONCAT(prc_path, '_dock_1_pick_available_led'), 
		process						:= prc, 
		CONVERSION_this				:= dock_1_pick_available_led);	

	led_init(
		object_name					:= CONCAT(prc_path, '_dock_1_AMR_ready_to_receive_led'), 
		process						:= prc, 
		CONVERSION_this				:= dock_1_AMR_ready_to_receive_led);	

	led_init(
		object_name					:= CONCAT(prc_path, '_dock_1_pick_location_conveyor_energized_led'), 
		process						:= prc, 
		CONVERSION_this				:= dock_1_pick_location_conveyor_energized_led);	

	led_init(
		object_name					:= CONCAT(prc_path, '_dock_2_drop_available_led'), 
		process						:= prc, 
		CONVERSION_this				:= dock_2_drop_available_led);	

	led_init(
		object_name					:= CONCAT(prc_path, '_dock_2_pick_available_led'), 
		process						:= prc, 
		CONVERSION_this				:= dock_2_pick_available_led);	

	led_init(
		object_name					:= CONCAT(prc_path, '_dock_2_AMR_ready_to_receive_led'), 
		process						:= prc, 
		CONVERSION_this				:= dock_2_AMR_ready_to_receive_led);	

	led_init(
		object_name					:= CONCAT(prc_path, '_dock_2_pick_location_conveyor_energized_led'), 
		process						:= prc, 
		CONVERSION_this				:= dock_2_pick_location_conveyor_energized_led);	
 	
	led_init(
		object_name					:= CONCAT(prc_path, '_ctCall_low_cup_supply_led'), 
		process						:= prc, 
		CONVERSION_this				:= ctCall_low_cup_supply_led);

	led_init(
		object_name					:= CONCAT(prc_path, '_ctCall_low_disk_supply_led'), 
		process						:= prc, 
		CONVERSION_this				:= ctCall_low_disk_supply_led);		

	led_init(
		object_name					:= CONCAT(prc_path, '_ctCall_low_lid_supply_led'), 
		process						:= prc, 
		CONVERSION_this				:= ctCall_low_lid_supply_led);	

	led_init(
		object_name					:= CONCAT(prc_path, '_ctCall_low_filter_supply_led'), 
		process						:= prc, 
		CONVERSION_this				:= ctCall_low_filter_supply_led);	

	led_init(
		object_name					:= CONCAT(prc_path, '_ctCall_scrap_full_led'), 
		process						:= prc, 
		CONVERSION_this				:= ctCall_scrap_full_led);	

	led_init(
		object_name					:= CONCAT(prc_path, '_ctCall_main_fault_led'), 
		process						:= prc, 
		CONVERSION_this				:= ctCall_main_fault_led);	

	led_init(
		object_name					:= CONCAT(prc_path, '_ctCall_cup_automation_fault_led'), 
		process						:= prc, 
		CONVERSION_this				:= ctCall_cup_automation_fault_led);	

	led_init(
		object_name					:= CONCAT(prc_path, '_ctCall_disk_automation_fault_led'), 
		process						:= prc, 
		CONVERSION_this				:= ctCall_disk_automation_fault_led);	

	led_init(
		object_name					:= CONCAT(prc_path, '_ctCall_lid_automation_fault_led'), 
		process						:= prc, 
		CONVERSION_this				:= ctCall_lid_automation_fault_led);	

	led_init(
		object_name					:= CONCAT(prc_path, '_ctCall_filter_automation_fault_led'), 
		process						:= prc, 
		CONVERSION_this				:= ctCall_filter_automation_fault_led);	
	
	parameter_overwrite_bool_init(
		object_name						:= CONCAT(prc_path, '_confirm_run_out_mode_pow'), 
		parameter						:= p_last_case, 
		process							:= prc, 
		CONVERSION_this					:= confirm_run_out_mode_pow);
		
	first_cycle := TRUE;		
		
END_IF

IF objects_running()
THEN
	process_cycle(prc);
END_IF
END_ACTION

ACTION _read_process_image:
;
END_ACTION

ACTION _read_var_input:
i_start_job_done 	:= ADR(csp_main_phaseManager_startJob.start_job_done);
END_ACTION

ACTION _set_runtime_properties:
;
END_ACTION

ACTION _write_output:
;
END_ACTION

ACTION custom_page:
hmi_graphic_object_set_status(
	status				:= HMI_OBJECT_STATUS_INVISIBLE, 
	CONVERSION_this		:= start_job_green_label);	

hmi_graphic_object_set_status(
	status				:= HMI_OBJECT_STATUS_INVISIBLE, 
	CONVERSION_this		:= steady_state_green_label);	
	
hmi_graphic_object_set_status(
	status				:= HMI_OBJECT_STATUS_INVISIBLE, 
	CONVERSION_this		:= cups_supply_green_label);

hmi_graphic_object_set_status(
	status				:= HMI_OBJECT_STATUS_INVISIBLE, 
	CONVERSION_this		:= carton_cases_supply_green_label);	
	
hmi_graphic_object_set_status(
	status				:= HMI_OBJECT_STATUS_INVISIBLE, 
	CONVERSION_this		:= production_green_label);	
	
hmi_graphic_object_set_status(
	status				:= HMI_OBJECT_STATUS_INVISIBLE, 
	CONVERSION_this		:= completion_green_label);	
	
hmi_graphic_object_set_status(
	status				:= HMI_OBJECT_STATUS_INVISIBLE, 
	CONVERSION_this		:= runout_green_label);

hmi_graphic_object_set_status(
	status				:= HMI_OBJECT_STATUS_INVISIBLE, 
	CONVERSION_this		:= end_job_green_label);

CASE fsm_status OF
	CSP_MAIN_PHASE_MANAGER_STATUS_START_JOB_10:
		hmi_graphic_object_set_status(
			status				:= HMI_OBJECT_STATUS_ON, 
			CONVERSION_this		:= start_job_green_label);
			
	CSP_MAIN_PHASE_MANAGER_STATUS_STEADY_STATE_20:
		hmi_graphic_object_set_status(
			status				:= HMI_OBJECT_STATUS_ON, 
			CONVERSION_this		:= steady_state_green_label);	
	
(*	CSP_MAIN_PHASE_MANAGER_STATUS_CUP_SUPPLY_30:
		hmi_graphic_object_set_status(
			status				:= HMI_OBJECT_STATUS_ON, 
			CONVERSION_this		:= cups_supply_green_label);	
	
	CSP_MAIN_PHASE_MANAGER_STATUS_CARTON_CASE_SUPPLY_40:
		hmi_graphic_object_set_status(
			status				:= HMI_OBJECT_STATUS_ON, 
			CONVERSION_this		:= carton_cases_supply_green_label);	*)
	
	CSP_MAIN_PHASE_MANAGER_MANUAL_STEADY_STATE_40:
		hmi_graphic_object_set_status(
			status				:= HMI_OBJECT_STATUS_ON, 
			CONVERSION_this		:= production_green_label);	
	
	CSP_MAIN_PHASE_MANAGER_STATUS_NEAR_END_OF_RUN_50:
		hmi_graphic_object_set_status(
			status				:= HMI_OBJECT_STATUS_ON, 
			CONVERSION_this		:= completion_green_label);	
	
	CSP_MAIN_PHASE_MANAGER_STATUS_RUNOUT_60:
		hmi_graphic_object_set_status(
			status				:= HMI_OBJECT_STATUS_ON, 
			CONVERSION_this		:= runout_green_label);	
	
	CSP_MAIN_PHASE_MANAGER_STATUS_END_JOB_70:
		hmi_graphic_object_set_status(
			status				:= HMI_OBJECT_STATUS_ON, 
			CONVERSION_this		:= end_job_green_label);	
ELSE
		hmi_graphic_object_set_status(
			status				:= HMI_OBJECT_STATUS_INVISIBLE, 
			CONVERSION_this		:= start_job_green_label);	

		hmi_graphic_object_set_status(
			status				:= HMI_OBJECT_STATUS_INVISIBLE, 
			CONVERSION_this		:= steady_state_green_label);	
			
		hmi_graphic_object_set_status(
			status				:= HMI_OBJECT_STATUS_INVISIBLE, 
			CONVERSION_this		:= cups_supply_green_label);
	
		hmi_graphic_object_set_status(
			status				:= HMI_OBJECT_STATUS_INVISIBLE, 
			CONVERSION_this		:= carton_cases_supply_green_label);	
			
		hmi_graphic_object_set_status(
			status				:= HMI_OBJECT_STATUS_INVISIBLE, 
			CONVERSION_this		:= production_green_label);	
			
		hmi_graphic_object_set_status(
			status				:= HMI_OBJECT_STATUS_INVISIBLE, 
			CONVERSION_this		:= completion_green_label);	
			
		hmi_graphic_object_set_status(
			status				:= HMI_OBJECT_STATUS_INVISIBLE, 
			CONVERSION_this		:= runout_green_label);
	
		hmi_graphic_object_set_status(
			status				:= HMI_OBJECT_STATUS_INVISIBLE, 
			CONVERSION_this		:= end_job_green_label);	
END_CASE

//LED update
IF machine_running
THEN
	led_set_color(
		color			:= HMI_LED_COLOR_GREEN, 
		CONVERSION_this	:= machine_running_led);
ELSE
	led_set_color(
		color			:= HMI_LED_COLOR_RED, 
		CONVERSION_this	:= machine_running_led);
END_IF

IF filler_faulted
THEN
	led_set_color(
		color			:= HMI_LED_COLOR_RED, 
		CONVERSION_this	:= filler_faulted_led);
ELSE
	led_set_color(
		color			:= HMI_LED_COLOR_GREEN, 
		CONVERSION_this	:= filler_faulted_led);
END_IF

IF filler_ready_for_coffee
THEN
	led_set_color(
		color			:= HMI_LED_COLOR_GREEN, 
		CONVERSION_this	:= ready_for_coffee_led);
ELSE
	led_set_color(
		color			:= HMI_LED_COLOR_RED, 
		CONVERSION_this	:= ready_for_coffee_led);
END_IF


IF cup_automation_faulted
THEN
	led_set_color(
		color			:= HMI_LED_COLOR_RED, 
		CONVERSION_this	:= cup_automation_faulted_led);
ELSE
	led_set_color(
		color			:= HMI_LED_COLOR_GREEN, 
		CONVERSION_this	:= cup_automation_faulted_led);
END_IF

IF disk_automation_faulted
THEN
	led_set_color(
		color			:= HMI_LED_COLOR_RED, 
		CONVERSION_this	:= disk_automation_faulted_led);
ELSE
	led_set_color(
		color			:= HMI_LED_COLOR_GREEN, 
		CONVERSION_this	:= disk_automation_faulted_led);
END_IF

IF filter_automation_faulted
THEN
	led_set_color(
		color			:= HMI_LED_COLOR_RED, 
		CONVERSION_this	:= filter_automation_faulted_led);
ELSE
	led_set_color(
		color			:= HMI_LED_COLOR_GREEN, 
		CONVERSION_this	:= filter_automation_faulted_led);
END_IF

IF lid_automation_faulted
THEN
	led_set_color(
		color			:= HMI_LED_COLOR_RED, 
		CONVERSION_this	:= lid_automation_faulted_led);
ELSE
	led_set_color(
		color			:= HMI_LED_COLOR_GREEN, 
		CONVERSION_this	:= lid_automation_faulted_led);
END_IF

IF emergency_stop_active
THEN
	led_set_color(
		color			:= HMI_LED_COLOR_RED, 
		CONVERSION_this	:= estop_active_led);
ELSE
	led_set_color(
		color			:= HMI_LED_COLOR_GREEN, 
		CONVERSION_this	:= estop_active_led);

END_IF

IF guard_open_stop_active
THEN
	led_set_color(
		color			:= HMI_LED_COLOR_RED, 
		CONVERSION_this	:= guard_open_led);
ELSE
	led_set_color(
		color			:= HMI_LED_COLOR_GREEN, 
		CONVERSION_this	:= guard_open_led);

END_IF

IF operator_stop_active
THEN
	led_set_color(
		color			:= HMI_LED_COLOR_RED, 
		CONVERSION_this	:= operator_stop_led);
ELSE
	led_set_color(
		color			:= HMI_LED_COLOR_GREEN, 
		CONVERSION_this	:= operator_stop_led);

END_IF

IF infeed_cups_missing
THEN
	led_set_color(
		color			:= HMI_LED_COLOR_RED, 
		CONVERSION_this	:= infeed_cups_missing_led);
ELSE
	led_set_color(
		color			:= HMI_LED_COLOR_GREEN, 
		CONVERSION_this	:= infeed_cups_missing_led);

END_IF

IF infeed_filters_missing
THEN
	led_set_color(
		color			:= HMI_LED_COLOR_RED, 
		CONVERSION_this	:= infeed_filters_missing_led);
ELSE
	led_set_color(
		color			:= HMI_LED_COLOR_GREEN, 
		CONVERSION_this	:= infeed_filters_missing_led);

END_IF

IF infeed_disks_missing
THEN
	led_set_color(
		color			:= HMI_LED_COLOR_RED, 
		CONVERSION_this	:= infeed_disks_missing_led);
ELSE
	led_set_color(
		color			:= HMI_LED_COLOR_GREEN, 
		CONVERSION_this	:= infeed_disks_missing_led);

END_IF

IF infeed_coffee_missing
THEN
	led_set_color(
		color			:= HMI_LED_COLOR_RED, 
		CONVERSION_this	:= infeed_coffee_missing_led);
ELSE
	led_set_color(
		color			:= HMI_LED_COLOR_GREEN, 
		CONVERSION_this	:= infeed_coffee_missing_led);

END_IF				
			
IF infeed_lids_missing
THEN
	led_set_color(
		color			:= HMI_LED_COLOR_RED, 
		CONVERSION_this	:= infeed_lids_missing_led);
ELSE
	led_set_color(
		color			:= HMI_LED_COLOR_GREEN, 
		CONVERSION_this	:= infeed_lids_missing_led);

END_IF	

IF downstream_block
THEN
	led_set_color(
		color			:= HMI_LED_COLOR_RED, 
		CONVERSION_this	:= downstream_block_led);
ELSE
	led_set_color(
		color			:= HMI_LED_COLOR_GREEN, 
		CONVERSION_this	:= downstream_block_led);

END_IF

IF reject_block
THEN
	led_set_color(
		color			:= HMI_LED_COLOR_RED, 
		CONVERSION_this	:= reject_block_led);
ELSE
	led_set_color(
		color			:= HMI_LED_COLOR_GREEN, 
		CONVERSION_this	:= reject_block_led);

END_IF

IF waste_block
THEN
	led_set_color(
		color			:= HMI_LED_COLOR_RED, 
		CONVERSION_this	:= waste_block_led);
ELSE
	led_set_color(
		color			:= HMI_LED_COLOR_GREEN, 
		CONVERSION_this	:= waste_block_led);

END_IF
		
IF csp_start_request
THEN
	led_set_color(
		color			:= HMI_LED_COLOR_GREEN, 
		CONVERSION_this	:= filler_start_request_led);
ELSE
	led_set_color(
		color			:= HMI_LED_COLOR_RED, 
		CONVERSION_this	:= filler_start_request_led);

END_IF

IF csp_start_ramp
THEN
	led_set_color(
		color			:= HMI_LED_COLOR_GREEN, 
		CONVERSION_this	:= filler_start_ramp_led);
ELSE
	led_set_color(
		color			:= HMI_LED_COLOR_RED, 
		CONVERSION_this	:= filler_start_ramp_led);

END_IF

IF csp_start_peak_wait
THEN
	led_set_color(
		color			:= HMI_LED_COLOR_RED, 
		CONVERSION_this	:= filler_start_peak_wait_led);
ELSE
	led_set_color(
		color			:= HMI_LED_COLOR_GREEN, 
		CONVERSION_this	:= filler_start_peak_wait_led);

END_IF

IF dock_1_drop_available
THEN
	led_set_color(
		color			:= HMI_LED_COLOR_GREEN, 
		CONVERSION_this	:= dock_1_drop_available_led);
ELSE
	led_set_color(
		color			:= HMI_LED_COLOR_YELLOW, 
		CONVERSION_this	:= dock_1_drop_available_led);

END_IF

IF dock_1_pick_available
THEN
	led_set_color(
		color			:= HMI_LED_COLOR_GREEN, 
		CONVERSION_this	:= dock_1_pick_available_led);
ELSE
	led_set_color(
		color			:= HMI_LED_COLOR_YELLOW, 
		CONVERSION_this	:= dock_1_pick_available_led);

END_IF

IF dock_1_AMR_ready_to_receive
THEN
	led_set_color(
		color			:= HMI_LED_COLOR_GREEN, 
		CONVERSION_this	:= dock_1_AMR_ready_to_receive_led);
ELSE
	led_set_color(
		color			:= HMI_LED_COLOR_GREY, 
		CONVERSION_this	:= dock_1_AMR_ready_to_receive_led);

END_IF

IF dock_1_pick_location_conveyor_energized
THEN
	led_set_color(
		color			:= HMI_LED_COLOR_GREEN, 
		CONVERSION_this	:= dock_1_pick_location_conveyor_energized_led);
ELSE
	led_set_color(
		color			:= HMI_LED_COLOR_GREY, 
		CONVERSION_this	:= dock_1_pick_location_conveyor_energized_led);

END_IF

IF dock_2_drop_available
THEN
	led_set_color(
		color			:= HMI_LED_COLOR_GREEN, 
		CONVERSION_this	:= dock_2_drop_available_led);
ELSE
	led_set_color(
		color			:= HMI_LED_COLOR_YELLOW, 
		CONVERSION_this	:= dock_2_drop_available_led);

END_IF

IF dock_2_pick_available
THEN
	led_set_color(
		color			:= HMI_LED_COLOR_GREEN, 
		CONVERSION_this	:= dock_2_pick_available_led);
ELSE
	led_set_color(
		color			:= HMI_LED_COLOR_YELLOW, 
		CONVERSION_this	:= dock_2_pick_available_led);

END_IF

IF dock_2_AMR_ready_to_receive
THEN
	led_set_color(
		color			:= HMI_LED_COLOR_GREEN, 
		CONVERSION_this	:= dock_2_AMR_ready_to_receive_led);
ELSE
	led_set_color(
		color			:= HMI_LED_COLOR_GREY, 
		CONVERSION_this	:= dock_2_AMR_ready_to_receive_led);

END_IF

IF dock_2_pick_location_conveyor_energized
THEN
	led_set_color(
		color			:= HMI_LED_COLOR_GREEN, 
		CONVERSION_this	:= dock_2_pick_location_conveyor_energized_led);
ELSE
	led_set_color(
		color			:= HMI_LED_COLOR_GREY, 
		CONVERSION_this	:= dock_2_pick_location_conveyor_energized_led);

END_IF












IF ctCall_low_cup_supply
THEN
	led_set_color(
		color			:= HMI_LED_COLOR_YELLOW, 
		CONVERSION_this	:= ctCall_low_cup_supply_led);
ELSE
	led_set_color(
		color			:= HMI_LED_COLOR_GREY, 
		CONVERSION_this	:= ctCall_low_cup_supply_led);

END_IF

IF ctCall_low_disk_supply
THEN
	led_set_color(
		color			:= HMI_LED_COLOR_YELLOW, 
		CONVERSION_this	:= ctCall_low_disk_supply_led);
ELSE
	led_set_color(
		color			:= HMI_LED_COLOR_GREY, 
		CONVERSION_this	:= ctCall_low_disk_supply_led);

END_IF

IF ctCall_low_lid_supply
THEN
	led_set_color(
		color			:= HMI_LED_COLOR_YELLOW, 
		CONVERSION_this	:= ctCall_low_lid_supply_led);
ELSE
	led_set_color(
		color			:= HMI_LED_COLOR_GREY, 
		CONVERSION_this	:= ctCall_low_lid_supply_led);

END_IF

IF ctCall_low_filter_supply
THEN
	led_set_color(
		color			:= HMI_LED_COLOR_YELLOW, 
		CONVERSION_this	:= ctCall_low_filter_supply_led);
ELSE
	led_set_color(
		color			:= HMI_LED_COLOR_GREY, 
		CONVERSION_this	:= ctCall_low_filter_supply_led);

END_IF

IF ctCall_scrap_full
THEN
	led_set_color(
		color			:= HMI_LED_COLOR_YELLOW, 
		CONVERSION_this	:= ctCall_scrap_full_led);
ELSE
	led_set_color(
		color			:= HMI_LED_COLOR_GREY, 
		CONVERSION_this	:= ctCall_scrap_full_led);

END_IF

IF ctCall_main_fault
THEN
	led_set_color(
		color			:= HMI_LED_COLOR_RED, 
		CONVERSION_this	:= ctCall_main_fault_led);
ELSE
	led_set_color(
		color			:= HMI_LED_COLOR_GREY, 
		CONVERSION_this	:= ctCall_main_fault_led);

END_IF

IF ctCall_cup_automation_fault
THEN
	led_set_color(
		color			:= HMI_LED_COLOR_RED, 
		CONVERSION_this	:= ctCall_cup_automation_fault_led);
ELSE
	led_set_color(
		color			:= HMI_LED_COLOR_GREY, 
		CONVERSION_this	:= ctCall_cup_automation_fault_led);

END_IF

IF ctCall_disk_automation_fault
THEN
	led_set_color(
		color			:= HMI_LED_COLOR_RED, 
		CONVERSION_this	:= ctCall_disk_automation_fault_led);
ELSE
	led_set_color(
		color			:= HMI_LED_COLOR_GREY, 
		CONVERSION_this	:= ctCall_disk_automation_fault_led);

END_IF

IF ctCall_lid_automation_fault
THEN
	led_set_color(
		color			:= HMI_LED_COLOR_RED, 
		CONVERSION_this	:= ctCall_lid_automation_fault_led);
ELSE
	led_set_color(
		color			:= HMI_LED_COLOR_GREY, 
		CONVERSION_this	:= ctCall_lid_automation_fault_led);

END_IF

IF ctCall_filter_automation_fault
THEN
	led_set_color(
		color			:= HMI_LED_COLOR_RED, 
		CONVERSION_this	:= ctCall_filter_automation_fault_led);
ELSE
	led_set_color(
		color			:= HMI_LED_COLOR_GREY, 
		CONVERSION_this	:= ctCall_filter_automation_fault_led);

END_IF
END_ACTION

ACTION run_cycle:
IF	csp_main.i_start_job_request
	AND	
	NOT csp_main.i_end_job_request
	AND
	NOT csp_main.i_cycle_enable_request
THEN
	fsm_status := CSP_MAIN_PHASE_MANAGER_STATUS_START_JOB_10;
END_IF

IF	NOT csp_main.i_start_job_request
	AND	csp_main.i_end_job_request
	AND
	NOT csp_main.i_cycle_enable_request
THEN
	fsm_status := CSP_MAIN_PHASE_MANAGER_STATUS_END_JOB_70;
END_IF


CASE fsm_status OF
	CSP_MAIN_PHASE_MANAGER_STATUS_UNDEFINED_0:
		start_MES_variables_update := FALSE;
		IF	p_mes_interface_enable
		THEN
			fsm_status := CSP_MAIN_PHASE_MANAGER_STATUS_START_JOB_10;
		ELSE
			fsm_status := CSP_MAIN_PHASE_MANAGER_MANUAL_STEADY_STATE_40;
		END_IF
		
	CSP_MAIN_PHASE_MANAGER_STATUS_START_JOB_10:
		start_MES_variables_update := FALSE;	
		IF csp_main_phaseManager_startJob.start_job_done
		THEN
			fsm_status := CSP_MAIN_PHASE_MANAGER_STATUS_STEADY_STATE_20;
		END_IF
		
	CSP_MAIN_PHASE_MANAGER_STATUS_STEADY_STATE_20:
		start_MES_variables_update := TRUE;
		i_start_job_done^ := FALSE;
		IF csp_main.i_cartoner_RunOutComplete //MARCO: to be added to CARTONER interface communication
		THEN
			fsm_status := CSP_MAIN_PHASE_MANAGER_STATUS_RUNOUT_60;
			//fsm_status := CSP_MAIN_PHASE_MANAGER_STATUS_NEAR_END_OF_RUN_50;
		END_IF
		
	CSP_MAIN_PHASE_MANAGER_STATUS_NEAR_END_OF_RUN_50:
		//IF 	csp_main_phaseManager_near_end_run.near_end_run_done //MARCO 1204
		//THEN
			fsm_status := CSP_MAIN_PHASE_MANAGER_STATUS_RUNOUT_60;
		//END_IF	

	CSP_MAIN_PHASE_MANAGER_STATUS_RUNOUT_60:
		IF	runout_completed
			AND
			NOT csp_main.i_cycle_enable_request
		THEN
			fsm_status := CSP_MAIN_PHASE_MANAGER_STATUS_END_JOB_70;
		END_IF	
		
	CSP_MAIN_PHASE_MANAGER_STATUS_END_JOB_70:
		IF	csp_main_phaseManager_end_job.end_job_done
		THEN	
			fsm_status := CSP_MAIN_PHASE_MANAGER_STATUS_UNDEFINED_0;
		END_IF
		
		
END_CASE
END_ACTION

ACTION variables_update:


bt_1sec(
	IN	:= (NOT bt_1sec_aux),
	PT	:= T#992MS,
	q	=> bt_1sec_aux);

IF	start_MES_variables_update
THEN

	IF	bt_1sec_aux
	THEN
		mes_elapsed_time_1_npr := mes_elapsed_time_1_npr + 1;
		
		IF	machine_is_running(csp.mch)	AND NOT csp_main_motorization_manager.suspend_conditions
		THEN
			 mes_elapsed_time_2_npr := mes_elapsed_time_2_npr + 1;
		END_IF
	END_IF

	IF machine_is_stopped(csp.mch)
    THEN
    	stop_message_CSP_ref := machine_get_downtime_stop_message(csp.mch);
    END_IF

	//Status update
	csp_main.i_csp_data_ref^.CaseBlanks.ConsumedCart 		:= 	0; 
	csp_main.i_csp_data_ref^.CaseBlanks.ConsumedTotal 		:= 	0;
	
	csp_main.i_csp_data_ref^.CtCall.FaultedCaseSupply		:= 	csp_case_feed_magazine.AML_Faulted;
	csp_main.i_csp_data_ref^.CtCall.FaultedMain				:= 	machine_is_stopped(csp.mch)
																AND 
																csp_main_interface.alarm_id <> 430 // SERVICE CYCLE STOP FOR CASE SIDE
																AND 
																csp_main_interface.alarm_id <> 431 // CYCLE STOP FOR CASE SIDE	
																AND 
																csp_main_interface.alarm_id <> 768 // SERVICE CYCLE STOP FOR TRANSFER SIDE
																AND 
																csp_main_interface.alarm_id <> 769;// CYCLE STOP FOR TRANSFER SIDE
																
	csp_main.i_csp_data_ref^.CtCall.FullScrapBin			:= 	message_is_on(csp_transfer_crosspusher_reject.backup_di_dchk.alarm_asm.message)
																OR
																message_is_on(csp_transfer_infeed_reject.bin_full_dchk.alarm_asm.message);
	csp_main.i_csp_data_ref^.CtCall.LowCaseSupply			:= 	csp_case_feed_magazine.AML_Robot_Out_Of_Cases; //MARCO - questo indica assenza Cases, non low_level
	csp_main.i_csp_data_ref^.CtCall.LowGlueSupply			:= 	NOT digital_input_is_active(csp_case_glue_hotmelt.level_ok_di);
	csp_main.i_csp_data_ref^.CtCall.LowLabelSupply			:= 	FALSE;//;inserire labeler presente nella Cartoner-step4
	csp_main.i_csp_data_ref^.CtCall.TBD1 					:= 	FALSE;
	csp_main.i_csp_data_ref^.CtCall.TBD2 					:= 	FALSE;	
	csp_main.i_csp_data_ref^.CtCall.TBD3 					:= 	FALSE;
	
	csp_main.i_csp_data_ref^.Production.GoodPods			:=	(
																	UDINT_TO_DINT(csp_case_main_statistics.logsect.hmi_shift_independent_sampled_counters.total_good_products)
																	*
																	csp_main_brand.case_pattern.case_pattern_L
																	*
																	csp_main_brand.case_pattern.case_pattern_W
																)
																*
																csp_main_brand.cups_number_for_carton;
																					
	csp_main.i_csp_data_ref^.Production.GoodUnits			:= 	UDINT_TO_DINT(csp_case_main_statistics.logsect.hmi_shift_independent_sampled_counters.total_good_products)
																*
																csp_main_brand.case_pattern.case_pattern_L
																*
																csp_main_brand.case_pattern.case_pattern_W;
																
	csp_main.i_csp_data_ref^.Production.GoodCases			:=	UDINT_TO_DINT(csp_case_main_statistics.logsect.hmi_shift_independent_sampled_counters.total_good_products);
	
	csp_main.i_csp_data_ref^.Production.GoodPodsNoReset		:=	(
																	UDINT_TO_DINT(csp_case_main_statistics.logsect.hmi_unresettable_sampled_counters.total_good_products)
																	*
																	csp_main_brand.case_pattern.case_pattern_L
																	*
																	csp_main_brand.case_pattern.case_pattern_W
																)
																*
																csp_main_brand.cups_number_for_carton;
	
